(* CoDeSys 2.3.9.41 project: gyps_plant.pro *)
(* Libraries: STANDARD.LIB 4.10.05 13:14:46, IECSFC.LIB 13.4.06 17:51:28, SYSLIBTIME.LIB 20.2.06 15:31:16, SYSTASKINFO.LIB 20.2.06 15:31:38, ANALYZATION.LIB 5.10.99 11:05:06, SYSLIBCALLBACK.LIB 20.2.06 15:31:08, Util.lib 18.5.10 17:14:28 *)

(* PLC configuration (modules and I/O channels)
Fast discrete inputs [I_SIMPLE_INPUT] node 0, in %IB0 out %QB0 {ChannellName = Fast discrete inputs; Filtrationtime = 10000}
  AT %IX0.0 [BitInput] Discrete input 1 {ChannellName = Enter name}
  AT %IX0.1 [BitInput] Discrete input 2 {ChannellName = Enter name}
  AT %IX0.2 [BitInput] Discrete input 3 {ChannellName = Enter name}
  AT %IX0.3 [BitInput] Discrete input 4 {ChannellName = Enter name}
Discrete inputs [ID130] node 1, in %IB1 out %QB1 {ChannellName = Discrete inputs; Filtrationtime_GeneralINP = 0; PinCount = 32}
  AT %IB1.0 [ByteInput] 8 discrete inputs {ChannellName = Enter name}
  AT %IB1.1 [ByteInput] 8 discrete inputs {ChannellName = Enter name}
  AT %IB1.2 [ByteInput] 8 discrete inputs {ChannellName = Enter name}
  AT %IB1.3 [ByteInput] 8 discrete inputs {ChannellName = Enter name}
AT %QX2.0 [BitOutput] Fast discrete output 1 {ChannellName = Enter name}
AT %QX2.1 [BitOutput] Fast discrete output 2 {ChannellName = Enter name}
AT %QX2.2 [BitOutput] Fast discrete output 3 {ChannellName = Enter name}
AT %QX2.3 [BitOutput] Fast discrete output 4 {ChannellName = Enter name}
Discrete outputs [ID131] node 3, in %IB3 out %QB3 {ChannellName = Discrete outputs; SafeValueByte = 0; SafeValueByte = 0; SafeValueByteM = 0; PinCount = 24}
  AT %QB3.0 [ByteOutput] 8 discrete outputs {ChannellName = Enter name}
  AT %QB3.1 [ByteOutput] 8 discrete outputs {ChannellName = Enter name}
  AT %QB3.2 [ByteOutput] 4 discrete outputs {ChannellName = Enter name}
Special input [ID103] node 4, in %IB4 out %QB4 {ChannellName = Special input}
  AT %IX4.0 [BitInput] Special input {ChannellName = Enter name}
Special output [ID104] node 5, in %IB5 out %QB5 {ChannellName = Special output}
  AT %QX5.0 [BitOutput] Special output {ChannellName = Enter name}
ModBus (Master) [MODBUS_MASTER_ID450] node 6, in %IB6 out %QB6 {ChannellName = ModBus (Master); Visibility = No}
  AT %QD6.0 [DWordOutput] Last address {ChannellName = Enter name}
  AT %QW6.1 [WordOutput] Last error {ChannellName = Enter name}
  RS-485-1 [COM1_USART] node 0, in %IB6.0 out %QB6.0 {ChannellName = RS-485-1; CommunicationSpeed = 115200; Parity = NO PARITY CHECK; BitLength = 8 bits; StopLength = One stop bit; InterfaceType = RS485; FrameOriented = RTU; Timeout = 0; Visibility = No}
  Universal Modbus device [ID2000] node 1, in %IB6.1 out %QB6.1 {ChannellName = Universal Modbus device; ModuleIP = 10:0:0:223; ServiceTimeout = 150; TCPport = 502; NetMode = Serial; ModuleSlaveAddress = 8; RequestType = By poll time; PeriodOfService = 10; Visibility = No; RepeatCounter = 0; ByteSequence = Trace_mode}
    AT %QB6.1.0 [ComChannel] Command (0xff - Start) {ChannellName = Enter name}
MV8_0 AT %QW6.1.0.0 [WordOutput] {ChannellName = Enter name}
MV8_1 AT %QW6.1.1.0 [WordOutput] {ChannellName = Enter name}
Universal Modbus device [ID2000] node 2, in %IB6.2 out %QB6.2 {ChannellName = Universal Modbus device; ModuleIP = 10:0:0:223; ServiceTimeout = 150; TCPport = 502; NetMode = Serial; ModuleSlaveAddress = 16; RequestType = By poll time; PeriodOfService = 10; Visibility = No; RepeatCounter = 0; ByteSequence = Trace_mode}
  AT %QB6.2.0 [ComChannel] Command (0xff - Start) {ChannellName = Enter name}
MV16_0 AT %QW6.2.0.0 [WordOutput] {ChannellName = Enter name}
Universal Modbus device [ID2000] node 3, in %IB6.3 out %QB6.3 {ChannellName = Universal Modbus device; ModuleIP = 10:0:0:223; ServiceTimeout = 150; TCPport = 502; NetMode = Serial; ModuleSlaveAddress = 24; RequestType = By poll time; PeriodOfService = 10; Visibility = No; RepeatCounter = 0; ByteSequence = Trace_mode}
  AT %QB6.3.0 [ComChannel] Command (0xff - Start) {ChannellName = Enter name}
MV24_0 AT %QW6.3.0.0 [WordOutput] {ChannellName = Enter name}
MV24_1 AT %QW6.3.1.0 [WordOutput] {ChannellName = Enter name}
Universal Modbus device [ID2000] node 4, in %IB6.4 out %QB6.4 {ChannellName = Universal Modbus device; ModuleIP = 10:0:0:223; ServiceTimeout = 150; TCPport = 502; NetMode = Serial; ModuleSlaveAddress = 32; RequestType = By poll time; PeriodOfService = 10; Visibility = No; RepeatCounter = 0; ByteSequence = Trace_mode}
  AT %QB6.4.0 [ComChannel] Command (0xff - Start) {ChannellName = Enter name}
MU01 AT %QW6.4.0.0 [WordOutput] {ChannellName = Enter name}
MU02 AT %QW6.4.1.0 [WordOutput] {ChannellName = Enter name}
MU03 AT %QW6.4.2.0 [WordOutput] {ChannellName = Enter name}
MU04 AT %QW6.4.3.0 [WordOutput] {ChannellName = Enter name}
MU05 AT %QW6.4.4.0 [WordOutput] {ChannellName = Enter name}
MU06 AT %QW6.4.5.0 [WordOutput] {ChannellName = Enter name}
MU07 AT %QW6.4.6.0 [WordOutput] {ChannellName = Enter name}
MU08 AT %QW6.4.7.0 [WordOutput] {ChannellName = Enter name}
MU09 AT %QW6.4.8.0 [WordOutput] {ChannellName = Enter name}
MU10 AT %QW6.4.9.0 [WordOutput] {ChannellName = Enter name}
MU11 AT %QW6.4.10.0 [WordOutput] {ChannellName = Enter name}
MU12 AT %QW6.4.11.0 [WordOutput] {ChannellName = Enter name}
MU13 AT %QW6.4.12.0 [WordOutput] {ChannellName = Enter name}
MU14 AT %QW6.4.13.0 [WordOutput] {ChannellName = Enter name}
MU15 AT %QW6.4.14.0 [WordOutput] {ChannellName = Enter name}
MU16 AT %QW6.4.15.0 [WordOutput] {ChannellName = Enter name}
MU17 AT %QW6.4.16.0 [WordOutput] {ChannellName = Enter name}
MU18 AT %QW6.4.17.0 [WordOutput] {ChannellName = Enter name}
MU19 AT %QW6.4.18.0 [WordOutput] {ChannellName = Enter name}
MU20 AT %QW6.4.19.0 [WordOutput] {ChannellName = Enter name}
MU21 AT %QW6.4.20.0 [WordOutput] {ChannellName = Enter name}
%MMU22 AT %QW6.4.21.0 [WordOutput] {ChannellName = Enter name}
MU23 AT %QW6.4.22.0 [WordOutput] {ChannellName = Enter name}
MU24 AT %QW6.4.23.0 [WordOutput] {ChannellName = Enter name}
MU25 AT %QW6.4.24.0 [WordOutput] {ChannellName = Enter name}
MU26 AT %QW6.4.25.0 [WordOutput] {ChannellName = Enter name}
MU27 AT %QW6.4.26.0 [WordOutput] {ChannellName = Enter name}
MU28 AT %QW6.4.27.0 [WordOutput] {ChannellName = Enter name}
MU29 AT %QW6.4.28.0 [WordOutput] {ChannellName = Enter name}
MU30 AT %QW6.4.29.0 [WordOutput] {ChannellName = Enter name}
MU31 AT %QW6.4.30.0 [WordOutput] {ChannellName = Enter name}
MU32 AT %QW6.4.31.0 [WordOutput] {ChannellName = Enter name}
AT %QB6.5.0 [ComChannel] Command (0xff - Start) {ChannellName = Enter name}
ELV_CURRENT_4 AT %QD6.5.0.0 [FloatOutput] {ChannellName = Enter name}
SHNK_CURRENT_4 AT %QD6.5.1.0 [FloatOutput] {ChannellName = Enter name}
MILL_SUCTION_4 AT %QD6.5.2.0 [FloatOutput] {ChannellName = Enter name}
SHNK_CURRENT_3 AT %QD6.5.3.0 [FloatOutput] {ChannellName = Enter name}
MILL_SUCTION_3 AT %QD6.5.4.0 [FloatOutput] {ChannellName = Enter name}
Universal Modbus device [ID2000] node 6, in %IB6.6 out %QB6.6 {ChannellName = Universal Modbus device; ModuleIP = 10:0:0:223; ServiceTimeout = 150; TCPport = 502; NetMode = Serial; ModuleSlaveAddress = 48; RequestType = By poll time; PeriodOfService = 10; Visibility = No; RepeatCounter = 0; ByteSequence = Trace_mode}
  AT %QB6.6.0 [ComChannel] Command (0xff - Start) {ChannellName = Enter name}
MV48_0 AT %QW6.6.0.0 [WordOutput] {ChannellName = Enter name}
MV48_1 AT %QW6.6.1.0 [WordOutput] {ChannellName = Enter name}
AT %QB6.7.0 [ComChannel] Command (0xff - Start) {ChannellName = Enter name}
ELV_CUR_0 AT %QD6.7.0.0 [FloatOutput] {ChannellName = Enter name}
SHOK_DROB_1 AT %QD6.7.1.0 [FloatOutput] {ChannellName = Enter name}
SHOK_DROB_2 AT %QD6.7.2.0 [FloatOutput] {ChannellName = Enter name}
ModBus (slave) [MODBUS_ID400] node 7, in %IB7 out %QB7 {ChannellName = ModBus (slave); SlaveIdentificator = 1; Visibility = No}
  Modbus [MODBUS_ID302] node 0, in %IB7.0 out %QB7.0 {ChannellName = Modbus}
    TCP [TCP_ID221] node 0, in %IB7.0.0 out %QB7.0.0 {ChannellName = TCP; RemotePort = 502; Visibility = No}
    TCP [TCP_ID221] node 1, in %IB7.0.1 out %QB7.0.1 {ChannellName = TCP; RemotePort = 503; Visibility = No}
  8 bits [8Bit] node 1, in %IB7.1 out %QB7.1 {ChannellName = 8 bit}
    REG_1_0 AT %QB7.1.0 [ByteOutput] {ChannellName = Enter name}
  8 bits [8Bit] node 2, in %IB7.2 out %QB7.2 {ChannellName = 8 bit}
    REG_1_1 AT %QB7.2.0 [ByteOutput] {ChannellName = Enter name}
  8 bits [8Bit] node 3, in %IB7.3 out %QB7.3 {ChannellName = 8 bit}
    REG_2_0 AT %QB7.3.0 [ByteOutput] {ChannellName = Enter name}
    REG_2_1 AT %QB7.4.0 [ByteOutput] {ChannellName = Enter name}
  8 bits [8Bit] node 5, in %IB7.5 out %QB7.5 {ChannellName = 8 bit}
    REG_3_0 AT %QB7.5.0 [ByteOutput] {ChannellName = Enter name}
  8 bits [8Bit] node 6, in %IB7.6 out %QB7.6 {ChannellName = 8 bit}
    REG_3_1 AT %QB7.6.0 [ByteOutput] {ChannellName = Enter name}
  8 bits [8Bit] node 7, in %IB7.7 out %QB7.7 {ChannellName = 8 bit}
    REG_4_0 AT %QB7.7.0 [ByteOutput] {ChannellName = Enter name}
    REG_4_1 AT %QB7.8.0 [ByteOutput] {ChannellName = Enter name}
    REG_5_0 AT %QB7.9.0 [ByteOutput] {ChannellName = Enter name}
  8 bits [8Bit] node 10, in %IB7.10 out %QB7.10 {ChannellName = 8 bit}
    REG_5_1 AT %QB7.10.0 [ByteOutput] {ChannellName = Enter name}
  8 bits [8Bit] node 11, in %IB7.11 out %QB7.11 {ChannellName = 8 bit}
    REG_6_0 AT %QB7.11.0 [ByteOutput] {ChannellName = Enter name}
    REG_6_1 AT %QB7.12.0 [ByteOutput] {ChannellName = Enter name}
  8 bits [8Bit] node 13, in %IB7.13 out %QB7.13 {ChannellName = 8 bit}
    REG_7_0 AT %QB7.13.0 [ByteOutput] {ChannellName = Enter name}
  8 bits [8Bit] node 14, in %IB7.14 out %QB7.14 {ChannellName = 8 bit}
    REG_7_1 AT %QB7.14.0 [ByteOutput] {ChannellName = Enter name}
  8 bits [8Bit] node 15, in %IB7.15 out %QB7.15 {ChannellName = 8 bit}
    REG_8_0 AT %QB7.15.0 [ByteOutput] {ChannellName = Enter name}
    REG_8_1 AT %QB7.16.0 [ByteOutput] {ChannellName = Enter name}
  8 bits [8Bit] node 17, in %IB7.17 out %QB7.17 {ChannellName = 8 bit}
    REG_9_0 AT %QB7.17.0 [ByteOutput] {ChannellName = Enter name}
  8 bits [8Bit] node 18, in %IB7.18 out %QB7.18 {ChannellName = 8 bit}
    REG_9_1 AT %QB7.18.0 [ByteOutput] {ChannellName = Enter name}
  8 bits [8Bit] node 19, in %IB7.19 out %QB7.19 {ChannellName = 8 bit}
    REG_10_0 AT %QB7.19.0 [ByteOutput] {ChannellName = Enter name}
    REG_10_1 AT %QB7.20.0 [ByteOutput] {ChannellName = Enter name}
  8 bits [8Bit] node 21, in %IB7.21 out %QB7.21 {ChannellName = 8 bit}
    REG_11_0 AT %QB7.21.0 [ByteOutput] {ChannellName = Enter name}
  8 bits [8Bit] node 22, in %IB7.22 out %QB7.22 {ChannellName = 8 bit}
    REG_11_1 AT %QB7.22.0 [ByteOutput] {ChannellName = Enter name}
  8 bits [8Bit] node 23, in %IB7.23 out %QB7.23 {ChannellName = 8 bit}
    REG_12_0 AT %QB7.23.0 [ByteOutput] {ChannellName = Enter name}
    REG_12_1 AT %QB7.24.0 [ByteOutput] {ChannellName = Enter name}
REG_13_ELV_CURRENT_4 AT %QD7.25.0 [FloatOutput] {ChannellName = Enter name}
REG_15_SHNK_CURRENT_4 AT %QD7.26.0 [FloatOutput] {ChannellName = Enter name}
REG_17_MILL_SUCTION_4 AT %QD7.27.0 [FloatOutput] {ChannellName = Enter name}
REG_19_SHNK_CURRENT_3 AT %QD7.28.0 [FloatOutput] {ChannellName = Enter name}
REG_21_MILL_SUCTION_3 AT %QD7.29.0 [FloatOutput] {ChannellName = Enter name}
REG_23_ELV_CUR_0 AT %QD7.30.0 [FloatOutput] {ChannellName = Enter name}
REG_25_SHOK_DROB_1 AT %QD7.31.0 [FloatOutput] {ChannellName = Enter name}
REG_27_SHOK_DROB_2 AT %QD7.32.0 [FloatOutput] {ChannellName = Enter name}
REG_29 AT %QD7.33.0 [FloatOutput] {ChannellName = Enter name}
REG_31 AT %QD7.34.0 [FloatOutput] {ChannellName = Enter name}
REG_33 AT %QD7.35.0 [FloatOutput] {ChannellName = Enter name}
REG_35 AT %QD7.36.0 [FloatOutput] {ChannellName = Enter name}
AT %QD8.0 [DWordOutput] Last address {ChannellName = Enter name}
AT %QW8.1 [WordOutput] Last error {ChannellName = Enter name}
RS-485-2 [COM3_USART] node 0, in %IB8.0 out %QB8.0 {ChannellName = RS-485-2; CommunicationSpeed = 115200; Parity = NO PARITY CHECK; BitLength = 8 bits; StopLength = One stop bit; InterfaceType = RS485; FrameOriented = RTU; Timeout = 0; Visibility = No}
Universal Modbus device [ID2000] node 1, in %IB8.1 out %QB8.1 {ChannellName = Universal Modbus device; ModuleIP = 10:0:0:223; ServiceTimeout = 150; TCPport = 502; NetMode = Serial; ModuleSlaveAddress = 1; RequestType = By poll time; PeriodOfService = 100; Visibility = No; RepeatCounter = 0; ByteSequence = Trace_mode}
  AT %QB8.1.0 [ComChannel] Command (0xff - Start) {ChannellName = Enter name}
CONV_PANEL_3 AT %QW8.1.0.0 [WordOutput] {ChannellName = Enter name}
CONV_FREQ_3 AT %QW8.1.1.0 [WordOutput] {ChannellName = Enter name}
CONV_CURRENT_3 AT %QW8.1.2.0 [WordOutput] {ChannellName = Enter name}
CONV_SET_FREQ_3 AT %QW8.1.3.0 [WordOutput] {ChannellName = Enter name}
AT %QB8.2.0 [ComChannel] Command (0xff - Start)
FAN_PANEL_3 AT %QW8.2.0.0 [WordOutput] {ChannellName = Enter name}
FAN_FREQ_3 AT %QW8.2.1.0 [WordOutput] {ChannellName = Enter name}
FAN_CURRENT_3 AT %QW8.2.2.0 [WordOutput] {ChannellName = Enter name}
FAN_SET_FREQ_3 AT %QW8.2.3.0 [WordOutput] {ChannellName = Enter name}
AT %QB8.3.0 [ComChannel] Command (0xff - Start) {ChannellName = Enter name}
MILL_PANEL_3 AT %QW8.3.0.0 [WordOutput] {ChannellName = Enter name}
MILL_FREQ_3 AT %QW8.3.1.0 [WordOutput] {ChannellName = Enter name}
MILL_CURRENT_3 AT %QW8.3.2.0 [WordOutput] {ChannellName = Enter name}
MILL_SET_FREQ_3 AT %QW8.3.3.0 [WordOutput] {ChannellName = Enter name}
AT %QB8.4.0 [ComChannel] Command (0xff - Start) {ChannellName = Enter name}
SEP_PANEL_3 AT %QW8.4.0.0 [WordOutput] {ChannellName = Enter name}
SEP_FREQ_3 AT %QW8.4.1.0 [WordOutput] {ChannellName = Enter name}
SEP_CURRENT_3 AT %QW8.4.2.0 [WordOutput] {ChannellName = Enter name}
SEP_SET_FREQ_3 AT %QW8.4.3.0 [WordOutput] {ChannellName = Enter name}
AT %QB8.5.0 [ComChannel] Command (0xff - Start) {ChannellName = Enter name}
CONV_PANEL_4 AT %QW8.5.0.0 [WordOutput] {ChannellName = Enter name}
CONV_FREQ_4 AT %QW8.5.1.0 [WordOutput] {ChannellName = Enter name}
CONV_CURRENT_4 AT %QW8.5.2.0 [WordOutput] {ChannellName = Enter name}
CONV_SET_FREQ_4 AT %QW8.5.3.0 [WordOutput] {ChannellName = Enter name}
AT %QB8.6.0 [ComChannel] Command (0xff - Start)
FAN_PANEL_4 AT %QW8.6.0.0 [WordOutput] {ChannellName = Enter name}
FAN_FREQ_4 AT %QW8.6.1.0 [WordOutput] {ChannellName = Enter name}
FAN_CURRENT_4 AT %QW8.6.2.0 [WordOutput] {ChannellName = Enter name}
FAN_SET_FREQ_4 AT %QW8.6.3.0 [WordOutput] {ChannellName = Enter name}
AT %QB8.7.0 [ComChannel] Command (0xff - Start) {ChannellName = Enter name}
MILL_PANEL_4 AT %QW8.7.0.0 [WordOutput] {ChannellName = Enter name}
MILL_FREQ_4 AT %QW8.7.1.0 [WordOutput] {ChannellName = Enter name}
MILL_CURRENT_4 AT %QW8.7.2.0 [WordOutput] {ChannellName = Enter name}
MILL_SET_FREQ_4 AT %QW8.7.3.0 [WordOutput] {ChannellName = Enter name}
AT %QB8.8.0 [ComChannel] Command (0xff - Start) {ChannellName = Enter name}
SEP_PANEL_4 AT %QW8.8.0.0 [WordOutput] {ChannellName = Enter name}
SEP_FREQ_4 AT %QW8.8.1.0 [WordOutput] {ChannellName = Enter name}
SEP_CURRENT_4 AT %QW8.8.2.0 [WordOutput] {ChannellName = Enter name}
SEP_SET_FREQ_4 AT %QW8.8.3.0 [WordOutput] {ChannellName = Enter name}
*)

(* Global variable list: Global_Variables *)
VAR_GLOBAL
	kvitVaqt : TIME := T#60s;
	tpKVIT : TP;
	HORN_RESET_0 : BOOL;
	(*MU 32 DISCRET OUTPUT*)
	ELV_RUN : BOOL;			(*DO01*)
	SHNK_RUN_4  : BOOL;		(*DO02*)
	SHNK_SKL_RUN_4  : BOOL;	(*DO03*)
	STAR_RUN_41  : BOOL;		(*DO04*)
	STAR_RUN_42  : BOOL;		(*DO05*)
	SEPR_RUN_4  : BOOL;		(*DO06*)
	OIL_ST_RUN_4  : BOOL;		(*DO07*)
	MILL_RUN_4  : BOOL;		(*DO08*)
	FAN_RUN_4  : BOOL;		(*DO09*)
	CONV_RUN_4  : BOOL;		(*DO10*)
	VIBR_RUN_4  : BOOL;		(*DO11*)
	VALV_RUN_4 : BOOL;		(*DO12*)
	HORN_RUN_4 : BOOL; 		(*DO13*)

	(*ELV_RUN_3 :  BOOL ; 		DO17*)
	SHNK_RUN_3 :  BOOL ; 		(*DO18*)
	SHNK_SKL_RUN_3 :  BOOL ; (*DO19*)
	STAR_RUN_31 :  BOOL ;  	(*DO20*)
	STAR_RUN_32 :  BOOL ;  	(*DO21*)
	SEPR_RUN_3 :  BOOL ;  		(*DO22*)
	OIL_ST_RUN_3 :  BOOL ;  	(*DO23*)
	MILL_RUN_3 :  BOOL ;  		(*DO24*)
	FAN_RUN_3 :  BOOL ;  		(*DO25*)
	CONV_RUN_3 :  BOOL ; 		(*DO26*)
	VIBR_RUN_3 :  BOOL ;  		(*DO27*)
	VALV_RUN_3 :  BOOL ;  		(*DO28*)
	HORN_RUN_3 :  BOOL ; 		(*DO29*)
	(*MU 32 DISCRET OUTPUT*)
	(*MV 24 DISCRET INPUT*)
	ELV_KM  : BOOL;				(*DI01*)
	SHNK_KM_4  : BOOL;			(*DI02*)
	SHNK_SKL_KM_4  : BOOL;		(*DI03*)
	STAR_KM_41  : BOOL;			(*DI04*)
	STAR_KM_42  : BOOL;			(*DI05*)
	SEPR_KM_4  : BOOL;			(*DI06*)
	OIL_ST_KM_4  : BOOL;			(*DI07*)
	MILL_KM_4  : BOOL;			(*DI08*)
	MATER_FULL_4  : BOOL;		(*DI09*)
	FAN_KM_4  : BOOL;				(*DI10*)
	CONV_KM_4  : BOOL;			(*DI11*)
	VIBR_KM_4  : BOOL;			(*DI12*)

				(*DI17*)
	SHNK_KM_3  : BOOL;			(*DI18*)
	SHNK_SKL_KM_3  : BOOL;		(*DI19*)
	STAR_KM_31  : BOOL;			(*DI20*)
	STAR_KM_32  : BOOL;			(*DI21*)
	SEPR_KM_3  : BOOL;			(*DI22*)
	OIL_ST_KM_3  : BOOL;			(*DI23*)
	MILL_KM_3  : BOOL;			(*DI24*)
	MATER_FULL_3  : BOOL;		(*DI25*)
	FAN_KM_3  : BOOL;				(*DI26*)
	CONV_KM_3  : BOOL;			(*DI27*)
	VIBR_KM_3  : BOOL;			(*DI28*)
	CONTR_PHASE_1_2 : BOOL;
	(*MV 24 DISCRET INPUT*)
	(*MV 16 DISCRET INPUT*)
	ELV_STOP_3  : BOOL;			(*DI01*)
	SHNK_STOP_3  : BOOL;			(*DI02*)
	SHNK_SKL_STOP_3  : BOOL;	(*DI03*)
	STAR_STOP_31  : BOOL;		(*DI04*)
	STAR_STOP_32  : BOOL;		(*DI05*)
	SEPR_STOP_3  : BOOL;			(*DI06*)
	OIL_ST_STOP_3  : BOOL;		(*DI07*)
	MILL_STOP_3  : BOOL;			(*DI08*)
	FAN_STOP_3  : BOOL;			(*DI09*)
	CONV_STOP_3  : BOOL;			(*DI10*)
	VIBR_STOP_3  : BOOL;			(*DI11*)

	ELV_START_3 : BOOL;			(*DI17*)
	SHNK_START_3 : BOOL;			(*DI18*)
	SHNK_SKL_START_3 : BOOL;	(*DI19*)
	STAR_START_31 : BOOL;		(*DI20*)
	STAR_START_32 : BOOL;		(*DI21*)
	SEPR_START_3 : BOOL;			(*DI22*)
	OIL_ST_START_3 : BOOL;		(*DI23*)
	MILL_START_3 : BOOL;			(*DI24*)
	FAN_START_3 : BOOL;			(*DI25*)
	CONV_START_3 : BOOL;		(*DI26*)
	VIBR_START_3 : BOOL;			(*DI27*)
	(*MV 16 DISCRET INPUT*)
	(*MV 08 DISCRET INPUT*)
	ELV_STOP_4  : BOOL;			(*DI01*)
	SHNK_STOP_4  : BOOL;			(*DI02*)
	SHNK_SKL_STOP_4  : BOOL;	(*DI03*)
	STAR_STOP_41  : BOOL;		(*DI04*)
	STAR_STOP_42  : BOOL;		(*DI05*)
	SEPR_STOP_4  : BOOL;			(*DI06*)
	OIL_ST_STOP_4  : BOOL;		(*DI07*)
	MILL_STOP_4  : BOOL;			(*DI08*)
	FAN_STOP_4  : BOOL;			(*DI09*)
	CONV_STOP_4  : BOOL;			(*DI10*)
	VIBR_STOP_4  : BOOL;			(*DI11*)

	ELV_START_4  : BOOL;			(*DI17*)
	SHNK_START_4  : BOOL;		(*DI18*)
	SHNK_SKL_START_4  : BOOL;	(*DI19*)
	STAR_START_41  : BOOL;		(*DI20*)
	STAR_START_42  : BOOL;		(*DI21*)
	SEPR_START_4  : BOOL;		(*DI22*)
	OIL_ST_START_4  : BOOL;		(*DI23*)
	MILL_START_4  : BOOL;			(*DI24*)
	FAN_START_4  : BOOL;			(*DI25*)
	CONV_START_4  : BOOL;			(*DI26*)
	VIBR_START_4  : BOOL;			(*DI27*)
	(*MV 08 DISCRET INPUT*)
END_VAR

(* Global variable list: mb_drob_in *)
VAR_GLOBAL
	MB_EMER_STOP_0 : BOOL;
	MB_MANUAL_ELV_0 : BOOL;
	MB_AUTO_ELV_0 : BOOL;
	MB_RESET_0 : BOOL;
	MB_ELV_STOP_0 : BOOL;
	MB_ELV_START_0 : BOOL;
	MB_SHOK_DROB_STOP_1 : BOOL;
	MB_SHOK_DROB_START_1 : BOOL;
	MB_SHOK_DROB_STOP_2 : BOOL;
	MB_SHOK_DROB_START_2 : BOOL;
	MB_CONV_STOP_0 : BOOL;
	MB_CONV_START_0 : BOOL;
	(****RESERV CONV ***)
	(***RESERV CONV****)
	MB_ELV_KM_0 : BOOL;
	MB_SHOK_DROB_KM_1 : BOOL;
	MB_SHOK_DROB_KM_2 : BOOL;
	MB_CONV_KM_0 : BOOL;
	(** RESERV KM CONV **)
	MB_TANK_MAX_0 : BOOL;
	MB_TANK_MIDLE_0 : BOOL;
	MB_TANK_MIN_0 : BOOL;


END_VAR

(* POU PLC_PRG, ST *)
PROGRAM PLC_PRG
VAR
END_VAR
main();
ALARMS();
RESET_ALRM();
TRANSLATE();
DROBILKA();
END_PROGRAM

(* POU main, LD *)
PROGRAM main
VAR
	MAH_YET3 : BOOL;
	VAQT : TIME := T#10s;
       VAQT1: TIME := T#4s;
       VAQT2 : TIME := T#6s;
      VAQT3 : TIME := T#6s;
	vaqtInduc : WORD := 15;
	VIBRATOR3_T: BOOL;
	TON1: TON;
	TON2: TON;
	OUT: BOOL;
	IND1: INDUKTIV;
	IND2: INDUKTIV;


	STOP: BOOL;
	CHIQSH: BOOL;
	PUSK: BOOL;
	MAH_YET4: BOOL;
	VIBRATOR4_T: BOOL;
	induk: BOOL;

	ALR_ELEV1: BOOL;
	ALR_ELEV2: BOOL;
	ALR_ELEV3: BOOL;
	ALR_ELEV4: BOOL;
	IND_ELV_1: INDUKTIV;
	IND_SHNK_3: INDUKTIV;
	IND_SHNK_4: INDUKTIV;
	IND_SHNK_SKL_4: INDUKTIV;
	IND_SEPR_4: INDUKTIV;
	IND_MILL_3: INDUKTIV;
	IND_MILL_4: INDUKTIV;

END_VAR
VAR (* helpers for the ST form of the networks *)
	_p1 : BOOL;
	_p2 : BOOL;
	_p3 : BOOL;
	_p4 : BOOL;
	_p5 : BOOL;
	_p6 : BOOL;
	_p7 : BOOL;
END_VAR
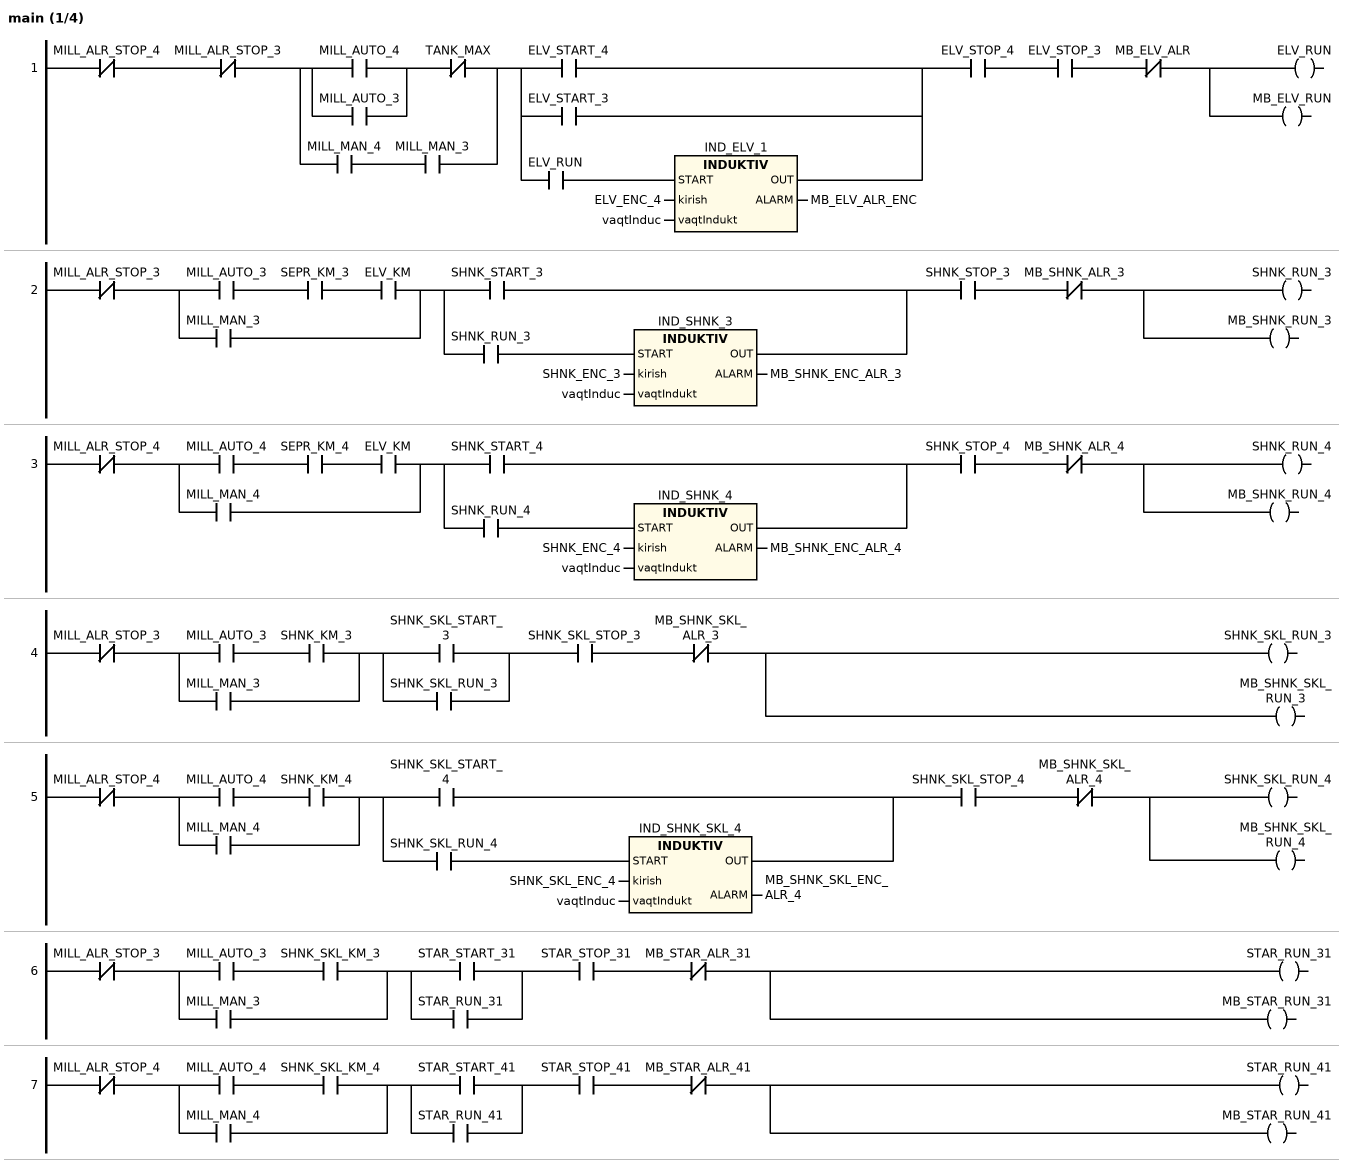
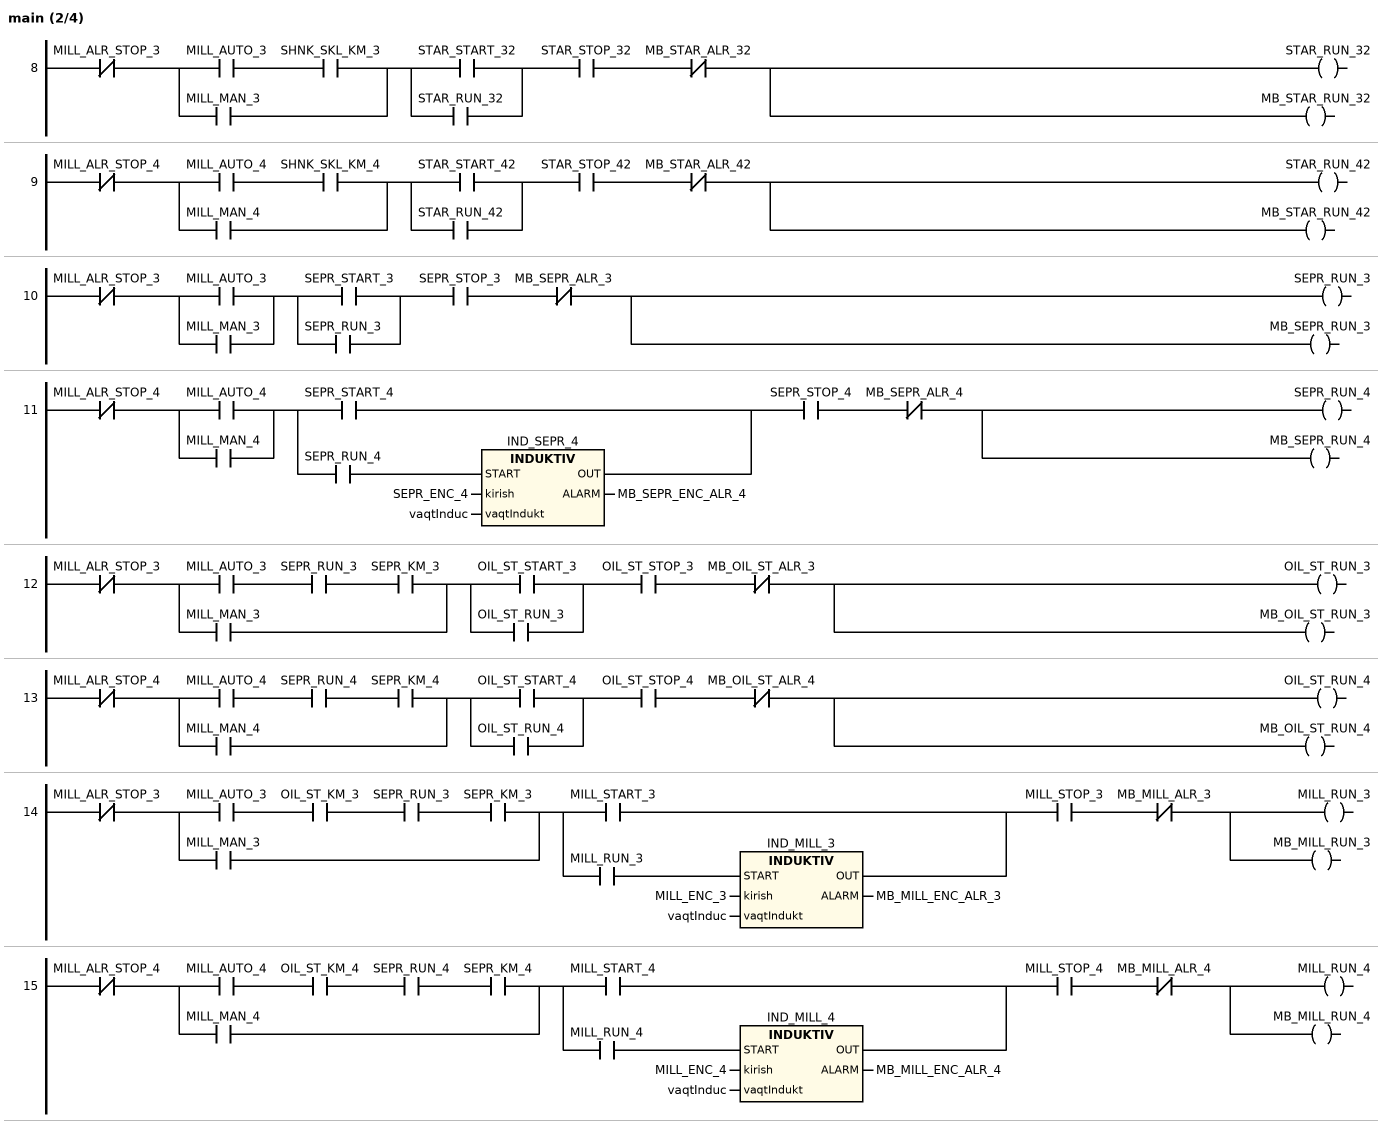
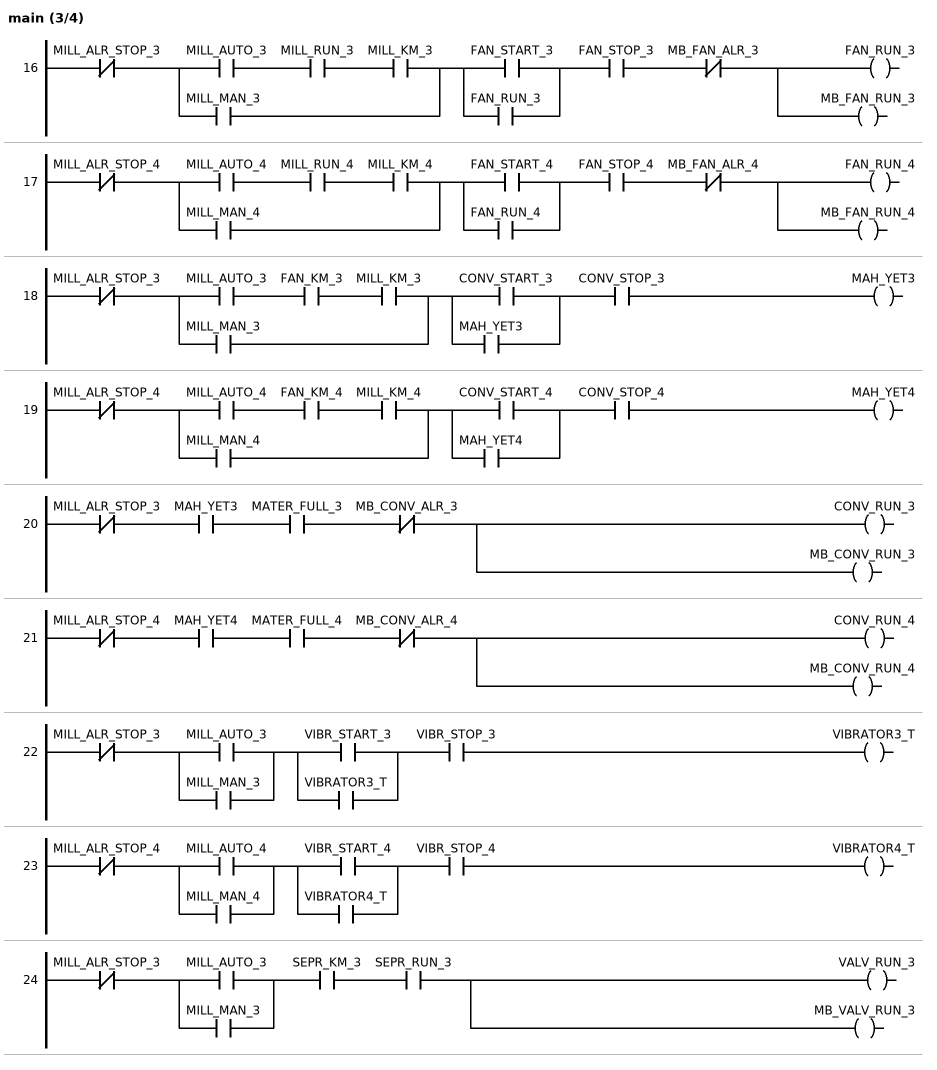
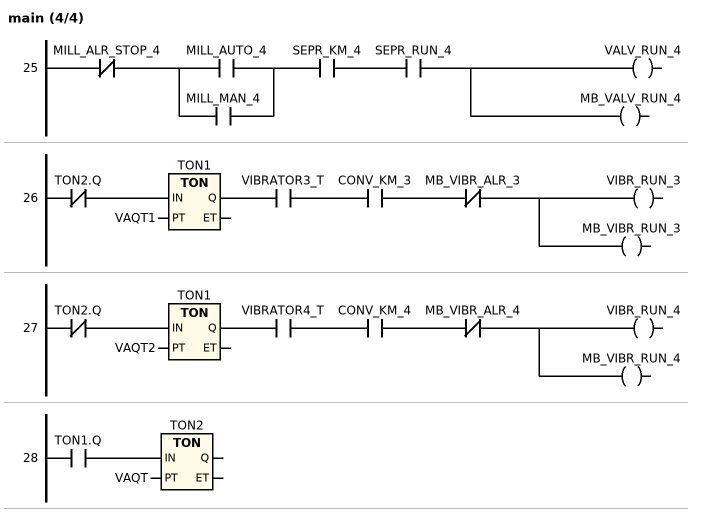
_LD_ (* Ladder Diagram *)
NETWORK 1
	[/MILL_ALR_STOP_4] - [/MILL_ALR_STOP_3] - { { [MILL_AUTO_4] | [MILL_AUTO_3] } - [/TANK_MAX] | [MILL_MAN_4] - [MILL_MAN_3] } - { [ELV_START_4] | [ELV_START_3] | [ELV_RUN] - IND_ELV_1:INDUKTIV(START: *, kirish: ELV_ENC_4, vaqtIndukt: vaqtInduc, ALARM => MB_ELV_ALR_ENC) } - [ELV_STOP_4] - [ELV_STOP_3] - [/MB_ELV_ALR] --- (ELV_RUN) (MB_ELV_RUN)
NETWORK 2
	[/MILL_ALR_STOP_3] - { [MILL_AUTO_3] - [SEPR_KM_3] - [ELV_KM] | [MILL_MAN_3] } - { [SHNK_START_3] | [SHNK_RUN_3] - IND_SHNK_3:INDUKTIV(START: *, kirish: SHNK_ENC_3, vaqtIndukt: vaqtInduc, ALARM => MB_SHNK_ENC_ALR_3) } - [SHNK_STOP_3] - [/MB_SHNK_ALR_3] --- (SHNK_RUN_3) (MB_SHNK_RUN_3)
NETWORK 3
	[/MILL_ALR_STOP_4] - { [MILL_AUTO_4] - [SEPR_KM_4] - [ELV_KM] | [MILL_MAN_4] } - { [SHNK_START_4] | [SHNK_RUN_4] - IND_SHNK_4:INDUKTIV(START: *, kirish: SHNK_ENC_4, vaqtIndukt: vaqtInduc, ALARM => MB_SHNK_ENC_ALR_4) } - [SHNK_STOP_4] - [/MB_SHNK_ALR_4] --- (SHNK_RUN_4) (MB_SHNK_RUN_4)
NETWORK 4
	[/MILL_ALR_STOP_3] - { [MILL_AUTO_3] - [SHNK_KM_3] | [MILL_MAN_3] } - { [SHNK_SKL_START_3] | [SHNK_SKL_RUN_3] } - [SHNK_SKL_STOP_3] - [/MB_SHNK_SKL_ALR_3] --- (SHNK_SKL_RUN_3) (MB_SHNK_SKL_RUN_3)
NETWORK 5
	[/MILL_ALR_STOP_4] - { [MILL_AUTO_4] - [SHNK_KM_4] | [MILL_MAN_4] } - { [SHNK_SKL_START_4] | [SHNK_SKL_RUN_4] - IND_SHNK_SKL_4:INDUKTIV(START: *, kirish: SHNK_SKL_ENC_4, vaqtIndukt: vaqtInduc, ALARM => MB_SHNK_SKL_ENC_ALR_4) } - [SHNK_SKL_STOP_4] - [/MB_SHNK_SKL_ALR_4] --- (SHNK_SKL_RUN_4) (MB_SHNK_SKL_RUN_4)
NETWORK 6
	[/MILL_ALR_STOP_3] - { [MILL_AUTO_3] - [SHNK_SKL_KM_3] | [MILL_MAN_3] } - { [STAR_START_31] | [STAR_RUN_31] } - [STAR_STOP_31] - [/MB_STAR_ALR_31] --- (STAR_RUN_31) (MB_STAR_RUN_31)
NETWORK 7
	[/MILL_ALR_STOP_4] - { [MILL_AUTO_4] - [SHNK_SKL_KM_4] | [MILL_MAN_4] } - { [STAR_START_41] | [STAR_RUN_41] } - [STAR_STOP_41] - [/MB_STAR_ALR_41] --- (STAR_RUN_41) (MB_STAR_RUN_41)
NETWORK 8
	[/MILL_ALR_STOP_3] - { [MILL_AUTO_3] - [SHNK_SKL_KM_3] | [MILL_MAN_3] } - { [STAR_START_32] | [STAR_RUN_32] } - [STAR_STOP_32] - [/MB_STAR_ALR_32] --- (STAR_RUN_32) (MB_STAR_RUN_32)
NETWORK 9
	[/MILL_ALR_STOP_4] - { [MILL_AUTO_4] - [SHNK_SKL_KM_4] | [MILL_MAN_4] } - { [STAR_START_42] | [STAR_RUN_42] } - [STAR_STOP_42] - [/MB_STAR_ALR_42] --- (STAR_RUN_42) (MB_STAR_RUN_42)
NETWORK 10
	[/MILL_ALR_STOP_3] - { [MILL_AUTO_3] | [MILL_MAN_3] } - { [SEPR_START_3] | [SEPR_RUN_3] } - [SEPR_STOP_3] - [/MB_SEPR_ALR_3] --- (SEPR_RUN_3) (MB_SEPR_RUN_3)
NETWORK 11
	[/MILL_ALR_STOP_4] - { [MILL_AUTO_4] | [MILL_MAN_4] } - { [SEPR_START_4] | [SEPR_RUN_4] - IND_SEPR_4:INDUKTIV(START: *, kirish: SEPR_ENC_4, vaqtIndukt: vaqtInduc, ALARM => MB_SEPR_ENC_ALR_4) } - [SEPR_STOP_4] - [/MB_SEPR_ALR_4] --- (SEPR_RUN_4) (MB_SEPR_RUN_4)
NETWORK 12
	[/MILL_ALR_STOP_3] - { [MILL_AUTO_3] - [SEPR_RUN_3] - [SEPR_KM_3] | [MILL_MAN_3] } - { [OIL_ST_START_3] | [OIL_ST_RUN_3] } - [OIL_ST_STOP_3] - [/MB_OIL_ST_ALR_3] --- (OIL_ST_RUN_3) (MB_OIL_ST_RUN_3)
NETWORK 13
	[/MILL_ALR_STOP_4] - { [MILL_AUTO_4] - [SEPR_RUN_4] - [SEPR_KM_4] | [MILL_MAN_4] } - { [OIL_ST_START_4] | [OIL_ST_RUN_4] } - [OIL_ST_STOP_4] - [/MB_OIL_ST_ALR_4] --- (OIL_ST_RUN_4) (MB_OIL_ST_RUN_4)
NETWORK 14
	[/MILL_ALR_STOP_3] - { [MILL_AUTO_3] - [OIL_ST_KM_3] - [SEPR_RUN_3] - [SEPR_KM_3] | [MILL_MAN_3] } - { [MILL_START_3] | [MILL_RUN_3] - IND_MILL_3:INDUKTIV(START: *, kirish: MILL_ENC_3, vaqtIndukt: vaqtInduc, ALARM => MB_MILL_ENC_ALR_3) } - [MILL_STOP_3] - [/MB_MILL_ALR_3] --- (MILL_RUN_3) (MB_MILL_RUN_3)
NETWORK 15
	[/MILL_ALR_STOP_4] - { [MILL_AUTO_4] - [OIL_ST_KM_4] - [SEPR_RUN_4] - [SEPR_KM_4] | [MILL_MAN_4] } - { [MILL_START_4] | [MILL_RUN_4] - IND_MILL_4:INDUKTIV(START: *, kirish: MILL_ENC_4, vaqtIndukt: vaqtInduc, ALARM => MB_MILL_ENC_ALR_4) } - [MILL_STOP_4] - [/MB_MILL_ALR_4] --- (MILL_RUN_4) (MB_MILL_RUN_4)
NETWORK 16
	[/MILL_ALR_STOP_3] - { [MILL_AUTO_3] - [MILL_RUN_3] - [MILL_KM_3] | [MILL_MAN_3] } - { [FAN_START_3] | [FAN_RUN_3] } - [FAN_STOP_3] - [/MB_FAN_ALR_3] --- (FAN_RUN_3) (MB_FAN_RUN_3)
NETWORK 17
	[/MILL_ALR_STOP_4] - { [MILL_AUTO_4] - [MILL_RUN_4] - [MILL_KM_4] | [MILL_MAN_4] } - { [FAN_START_4] | [FAN_RUN_4] } - [FAN_STOP_4] - [/MB_FAN_ALR_4] --- (FAN_RUN_4) (MB_FAN_RUN_4)
NETWORK 18
	[/MILL_ALR_STOP_3] - { [MILL_AUTO_3] - [FAN_KM_3] - [MILL_KM_3] | [MILL_MAN_3] } - { [CONV_START_3] | [MAH_YET3] } - [CONV_STOP_3] --- (MAH_YET3)
NETWORK 19
	[/MILL_ALR_STOP_4] - { [MILL_AUTO_4] - [FAN_KM_4] - [MILL_KM_4] | [MILL_MAN_4] } - { [CONV_START_4] | [MAH_YET4] } - [CONV_STOP_4] --- (MAH_YET4)
NETWORK 20
	[/MILL_ALR_STOP_3] - [MAH_YET3] - [MATER_FULL_3] - [/MB_CONV_ALR_3] --- (CONV_RUN_3) (MB_CONV_RUN_3)
NETWORK 21
	[/MILL_ALR_STOP_4] - [MAH_YET4] - [MATER_FULL_4] - [/MB_CONV_ALR_4] --- (CONV_RUN_4) (MB_CONV_RUN_4)
NETWORK 22
	[/MILL_ALR_STOP_3] - { [MILL_AUTO_3] | [MILL_MAN_3] } - { [VIBR_START_3] | [VIBRATOR3_T] } - [VIBR_STOP_3] --- (VIBRATOR3_T)
NETWORK 23
	[/MILL_ALR_STOP_4] - { [MILL_AUTO_4] | [MILL_MAN_4] } - { [VIBR_START_4] | [VIBRATOR4_T] } - [VIBR_STOP_4] --- (VIBRATOR4_T)
NETWORK 24
	[/MILL_ALR_STOP_3] - { [MILL_AUTO_3] | [MILL_MAN_3] } - [SEPR_KM_3] - [SEPR_RUN_3] --- (VALV_RUN_3) (MB_VALV_RUN_3)
NETWORK 25
	[/MILL_ALR_STOP_4] - { [MILL_AUTO_4] | [MILL_MAN_4] } - [SEPR_KM_4] - [SEPR_RUN_4] --- (VALV_RUN_4) (MB_VALV_RUN_4)
NETWORK 26
	[/TON2.Q] - TON1:TON(IN: *, PT: VAQT1) - [VIBRATOR3_T] - [CONV_KM_3] - [/MB_VIBR_ALR_3] --- (VIBR_RUN_3) (MB_VIBR_RUN_3)
NETWORK 27
	[/TON2.Q] - TON1:TON(IN: *, PT: VAQT2) - [VIBRATOR4_T] - [CONV_KM_4] - [/MB_VIBR_ALR_4] --- (VIBR_RUN_4) (MB_VIBR_RUN_4)
NETWORK 28
	[TON1.Q] - TON2:TON(IN: *, PT: VAQT)
_END_LD_
(* the same logic as Structured Text *)
(* Network 1 *)
_p1 := NOT MILL_ALR_STOP_4 AND NOT MILL_ALR_STOP_3 AND ((MILL_AUTO_4 OR MILL_AUTO_3) AND NOT TANK_MAX OR MILL_MAN_4 AND MILL_MAN_3);
IND_ELV_1(START := _p1 AND ELV_RUN, kirish := ELV_ENC_4, vaqtIndukt := vaqtInduc);
MB_ELV_ALR_ENC := IND_ELV_1.ALARM;
ELV_RUN := (_p1 AND ELV_START_4 OR _p1 AND ELV_START_3 OR IND_ELV_1.OUT) AND ELV_STOP_4 AND ELV_STOP_3 AND NOT MB_ELV_ALR;
MB_ELV_RUN := ELV_RUN;
(* Network 2 *)
_p2 := NOT MILL_ALR_STOP_3 AND (MILL_AUTO_3 AND SEPR_KM_3 AND ELV_KM OR MILL_MAN_3);
IND_SHNK_3(START := _p2 AND SHNK_RUN_3, kirish := SHNK_ENC_3, vaqtIndukt := vaqtInduc);
MB_SHNK_ENC_ALR_3 := IND_SHNK_3.ALARM;
SHNK_RUN_3 := (_p2 AND SHNK_START_3 OR IND_SHNK_3.OUT) AND SHNK_STOP_3 AND NOT MB_SHNK_ALR_3;
MB_SHNK_RUN_3 := SHNK_RUN_3;
(* Network 3 *)
_p3 := NOT MILL_ALR_STOP_4 AND (MILL_AUTO_4 AND SEPR_KM_4 AND ELV_KM OR MILL_MAN_4);
IND_SHNK_4(START := _p3 AND SHNK_RUN_4, kirish := SHNK_ENC_4, vaqtIndukt := vaqtInduc);
MB_SHNK_ENC_ALR_4 := IND_SHNK_4.ALARM;
SHNK_RUN_4 := (_p3 AND SHNK_START_4 OR IND_SHNK_4.OUT) AND SHNK_STOP_4 AND NOT MB_SHNK_ALR_4;
MB_SHNK_RUN_4 := SHNK_RUN_4;
(* Network 4 *)
SHNK_SKL_RUN_3 := NOT MILL_ALR_STOP_3 AND (MILL_AUTO_3 AND SHNK_KM_3 OR MILL_MAN_3) AND (SHNK_SKL_START_3 OR SHNK_SKL_RUN_3) AND SHNK_SKL_STOP_3 AND NOT MB_SHNK_SKL_ALR_3;
MB_SHNK_SKL_RUN_3 := SHNK_SKL_RUN_3;
(* Network 5 *)
_p4 := NOT MILL_ALR_STOP_4 AND (MILL_AUTO_4 AND SHNK_KM_4 OR MILL_MAN_4);
IND_SHNK_SKL_4(START := _p4 AND SHNK_SKL_RUN_4, kirish := SHNK_SKL_ENC_4, vaqtIndukt := vaqtInduc);
MB_SHNK_SKL_ENC_ALR_4 := IND_SHNK_SKL_4.ALARM;
SHNK_SKL_RUN_4 := (_p4 AND SHNK_SKL_START_4 OR IND_SHNK_SKL_4.OUT) AND SHNK_SKL_STOP_4 AND NOT MB_SHNK_SKL_ALR_4;
MB_SHNK_SKL_RUN_4 := SHNK_SKL_RUN_4;
(* Network 6 *)
STAR_RUN_31 := NOT MILL_ALR_STOP_3 AND (MILL_AUTO_3 AND SHNK_SKL_KM_3 OR MILL_MAN_3) AND (STAR_START_31 OR STAR_RUN_31) AND STAR_STOP_31 AND NOT MB_STAR_ALR_31;
MB_STAR_RUN_31 := STAR_RUN_31;
(* Network 7 *)
STAR_RUN_41 := NOT MILL_ALR_STOP_4 AND (MILL_AUTO_4 AND SHNK_SKL_KM_4 OR MILL_MAN_4) AND (STAR_START_41 OR STAR_RUN_41) AND STAR_STOP_41 AND NOT MB_STAR_ALR_41;
MB_STAR_RUN_41 := STAR_RUN_41;
(* Network 8 *)
STAR_RUN_32 := NOT MILL_ALR_STOP_3 AND (MILL_AUTO_3 AND SHNK_SKL_KM_3 OR MILL_MAN_3) AND (STAR_START_32 OR STAR_RUN_32) AND STAR_STOP_32 AND NOT MB_STAR_ALR_32;
MB_STAR_RUN_32 := STAR_RUN_32;
(* Network 9 *)
STAR_RUN_42 := NOT MILL_ALR_STOP_4 AND (MILL_AUTO_4 AND SHNK_SKL_KM_4 OR MILL_MAN_4) AND (STAR_START_42 OR STAR_RUN_42) AND STAR_STOP_42 AND NOT MB_STAR_ALR_42;
MB_STAR_RUN_42 := STAR_RUN_42;
(* Network 10 *)
SEPR_RUN_3 := NOT MILL_ALR_STOP_3 AND (MILL_AUTO_3 OR MILL_MAN_3) AND (SEPR_START_3 OR SEPR_RUN_3) AND SEPR_STOP_3 AND NOT MB_SEPR_ALR_3;
MB_SEPR_RUN_3 := SEPR_RUN_3;
(* Network 11 *)
_p5 := NOT MILL_ALR_STOP_4 AND (MILL_AUTO_4 OR MILL_MAN_4);
IND_SEPR_4(START := _p5 AND SEPR_RUN_4, kirish := SEPR_ENC_4, vaqtIndukt := vaqtInduc);
MB_SEPR_ENC_ALR_4 := IND_SEPR_4.ALARM;
SEPR_RUN_4 := (_p5 AND SEPR_START_4 OR IND_SEPR_4.OUT) AND SEPR_STOP_4 AND NOT MB_SEPR_ALR_4;
MB_SEPR_RUN_4 := SEPR_RUN_4;
(* Network 12 *)
OIL_ST_RUN_3 := NOT MILL_ALR_STOP_3 AND (MILL_AUTO_3 AND SEPR_RUN_3 AND SEPR_KM_3 OR MILL_MAN_3) AND (OIL_ST_START_3 OR OIL_ST_RUN_3) AND OIL_ST_STOP_3 AND NOT MB_OIL_ST_ALR_3;
MB_OIL_ST_RUN_3 := OIL_ST_RUN_3;
(* Network 13 *)
OIL_ST_RUN_4 := NOT MILL_ALR_STOP_4 AND (MILL_AUTO_4 AND SEPR_RUN_4 AND SEPR_KM_4 OR MILL_MAN_4) AND (OIL_ST_START_4 OR OIL_ST_RUN_4) AND OIL_ST_STOP_4 AND NOT MB_OIL_ST_ALR_4;
MB_OIL_ST_RUN_4 := OIL_ST_RUN_4;
(* Network 14 *)
_p6 := NOT MILL_ALR_STOP_3 AND (MILL_AUTO_3 AND OIL_ST_KM_3 AND SEPR_RUN_3 AND SEPR_KM_3 OR MILL_MAN_3);
IND_MILL_3(START := _p6 AND MILL_RUN_3, kirish := MILL_ENC_3, vaqtIndukt := vaqtInduc);
MB_MILL_ENC_ALR_3 := IND_MILL_3.ALARM;
MILL_RUN_3 := (_p6 AND MILL_START_3 OR IND_MILL_3.OUT) AND MILL_STOP_3 AND NOT MB_MILL_ALR_3;
MB_MILL_RUN_3 := MILL_RUN_3;
(* Network 15 *)
_p7 := NOT MILL_ALR_STOP_4 AND (MILL_AUTO_4 AND OIL_ST_KM_4 AND SEPR_RUN_4 AND SEPR_KM_4 OR MILL_MAN_4);
IND_MILL_4(START := _p7 AND MILL_RUN_4, kirish := MILL_ENC_4, vaqtIndukt := vaqtInduc);
MB_MILL_ENC_ALR_4 := IND_MILL_4.ALARM;
MILL_RUN_4 := (_p7 AND MILL_START_4 OR IND_MILL_4.OUT) AND MILL_STOP_4 AND NOT MB_MILL_ALR_4;
MB_MILL_RUN_4 := MILL_RUN_4;
(* Network 16 *)
FAN_RUN_3 := NOT MILL_ALR_STOP_3 AND (MILL_AUTO_3 AND MILL_RUN_3 AND MILL_KM_3 OR MILL_MAN_3) AND (FAN_START_3 OR FAN_RUN_3) AND FAN_STOP_3 AND NOT MB_FAN_ALR_3;
MB_FAN_RUN_3 := FAN_RUN_3;
(* Network 17 *)
FAN_RUN_4 := NOT MILL_ALR_STOP_4 AND (MILL_AUTO_4 AND MILL_RUN_4 AND MILL_KM_4 OR MILL_MAN_4) AND (FAN_START_4 OR FAN_RUN_4) AND FAN_STOP_4 AND NOT MB_FAN_ALR_4;
MB_FAN_RUN_4 := FAN_RUN_4;
(* Network 18 *)
MAH_YET3 := NOT MILL_ALR_STOP_3 AND (MILL_AUTO_3 AND FAN_KM_3 AND MILL_KM_3 OR MILL_MAN_3) AND (CONV_START_3 OR MAH_YET3) AND CONV_STOP_3;
(* Network 19 *)
MAH_YET4 := NOT MILL_ALR_STOP_4 AND (MILL_AUTO_4 AND FAN_KM_4 AND MILL_KM_4 OR MILL_MAN_4) AND (CONV_START_4 OR MAH_YET4) AND CONV_STOP_4;
(* Network 20 *)
CONV_RUN_3 := NOT MILL_ALR_STOP_3 AND MAH_YET3 AND MATER_FULL_3 AND NOT MB_CONV_ALR_3;
MB_CONV_RUN_3 := CONV_RUN_3;
(* Network 21 *)
CONV_RUN_4 := NOT MILL_ALR_STOP_4 AND MAH_YET4 AND MATER_FULL_4 AND NOT MB_CONV_ALR_4;
MB_CONV_RUN_4 := CONV_RUN_4;
(* Network 22 *)
VIBRATOR3_T := NOT MILL_ALR_STOP_3 AND (MILL_AUTO_3 OR MILL_MAN_3) AND (VIBR_START_3 OR VIBRATOR3_T) AND VIBR_STOP_3;
(* Network 23 *)
VIBRATOR4_T := NOT MILL_ALR_STOP_4 AND (MILL_AUTO_4 OR MILL_MAN_4) AND (VIBR_START_4 OR VIBRATOR4_T) AND VIBR_STOP_4;
(* Network 24 *)
VALV_RUN_3 := NOT MILL_ALR_STOP_3 AND (MILL_AUTO_3 OR MILL_MAN_3) AND SEPR_KM_3 AND SEPR_RUN_3;
MB_VALV_RUN_3 := VALV_RUN_3;
(* Network 25 *)
VALV_RUN_4 := NOT MILL_ALR_STOP_4 AND (MILL_AUTO_4 OR MILL_MAN_4) AND SEPR_KM_4 AND SEPR_RUN_4;
MB_VALV_RUN_4 := VALV_RUN_4;
(* Network 26 *)
TON1(IN := NOT TON2.Q, PT := VAQT1);
VIBR_RUN_3 := TON1.Q AND VIBRATOR3_T AND CONV_KM_3 AND NOT MB_VIBR_ALR_3;
MB_VIBR_RUN_3 := VIBR_RUN_3;
(* Network 27 *)
TON1(IN := NOT TON2.Q, PT := VAQT2);
VIBR_RUN_4 := TON1.Q AND VIBRATOR4_T AND CONV_KM_4 AND NOT MB_VIBR_ALR_4;
MB_VIBR_RUN_4 := VIBR_RUN_4;
(* Network 28 *)
TON2(IN := TON1.Q, PT := VAQT);
END_PROGRAM

(* POU INDUKTIV, CFC *)
FUNCTION_BLOCK INDUKTIV
VAR_IN_OUT

	(*RESET : BOOL;*)

END_VAR
VAR_INPUT
	START : BOOL;
	kirish : BOOL;
	vaqtIndukt : WORD := 15;
END_VAR

VAR_OUTPUT

	OUT : BOOL;
	ALARM : BOOL;
END_VAR
VAR
	ton1: TON;
	vaqt : TIME;
	ton2: TON;
	TP1: TP;
	TP2: TP;


END_VAR
VAR (* helpers for the ST form of the networks *)
	_t11 : BOOL;
	_t41 : BOOL;
	_t47 : BOOL;
END_VAR
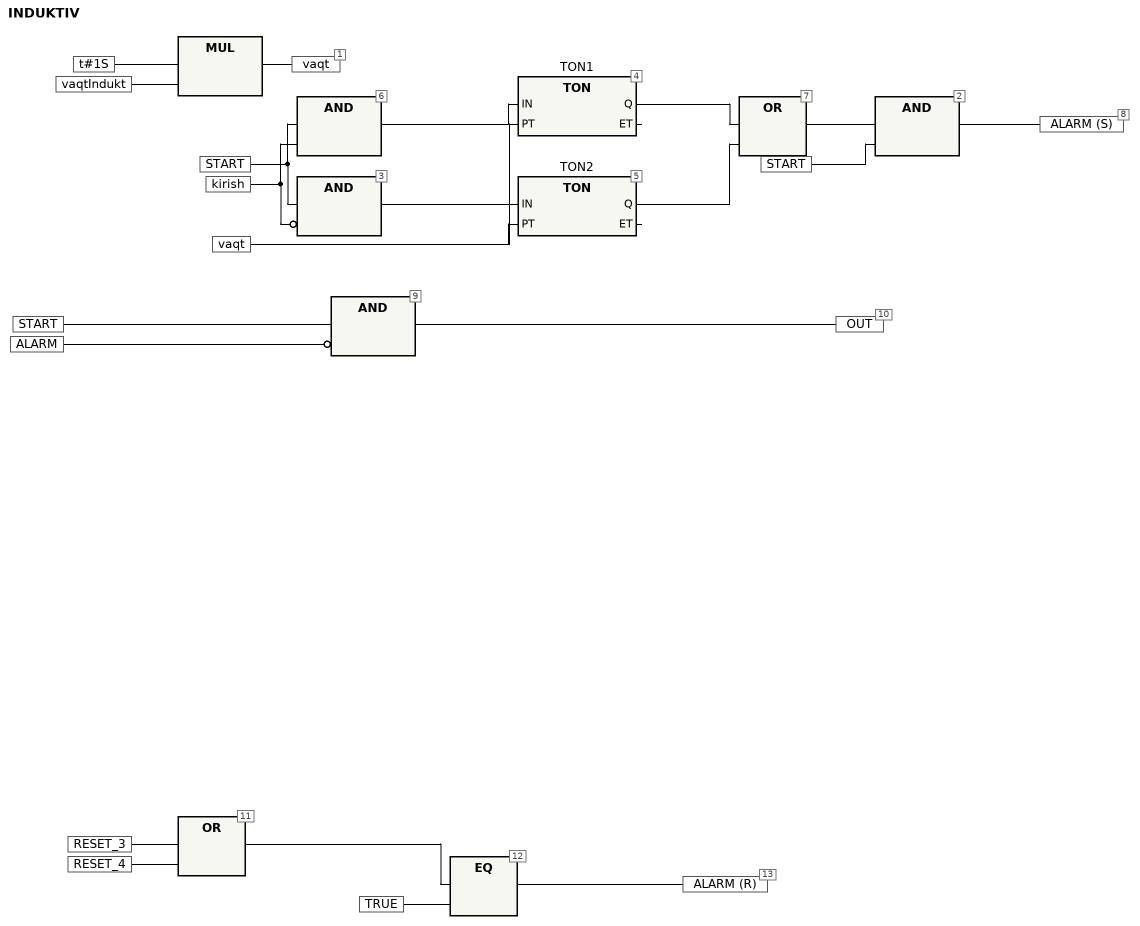
_CFC_ (* Continuous Function Chart, elements in execution order *)
#0 MUL(t#1S, vaqtIndukt)
#1 vaqt <= #0
#2 AND(#7, START)
#3 AND(START, NOT kirish)
#4 TON1:TON(IN: #6, PT: vaqt)
#5 TON2:TON(IN: #3, PT: vaqt)
#6 AND(START, kirish)
#7 OR(#4.Q, #5.Q)
#8 S ALARM <= #2
#9 AND(START, NOT ALARM)
#10 OUT <= #9
#11 OR(RESET_3, RESET_4)
#12 EQ(#11, TRUE)
#13 R ALARM <= #12
_END_CFC_
(* the same logic as Structured Text *)
vaqt := t#1S * vaqtIndukt;
_t41 := _t11 AND START;
TON1(IN := _t47, PT := vaqt);
TON2(IN := START AND NOT kirish, PT := vaqt);
_t47 := START AND kirish;
_t11 := TON1.Q OR TON2.Q;
IF _t41 THEN ALARM := TRUE; END_IF;
OUT := START AND NOT ALARM;
IF (RESET_3 OR RESET_4) = TRUE THEN ALARM := FALSE; END_IF;
END_FUNCTION_BLOCK

(* POU ALARMS, LD *)
PROGRAM ALARMS
VAR
	tofELV: TON;
	tofSHNK3: TON;
	tofSHNK4: TON;
	tofSHNK_SKL_3: TON;
	tofSHNK_SKL_4: TON;
	tofSTAR_31: TON;
	tofSTAR_32: TON;
	tofSTAR_41: TON;
	tofSTAR_42: TON;
	tofSEPR_3: TON;
	tofSEPR_4: TON;
	tofOIL_3: TON;
	tofOIL_4: TON;
	tofMILL_3: TON;
	tofMILL_4: TON;
	tofFAN_3: TON;
	tofFAN_4: TON;
	tofCONV_3: TON;
	tofCONV_4: TON;
	tofVIB_3: TON;
	tofVIB_4: TON;

	vaqt : TIME := T#30S;
END_VAR
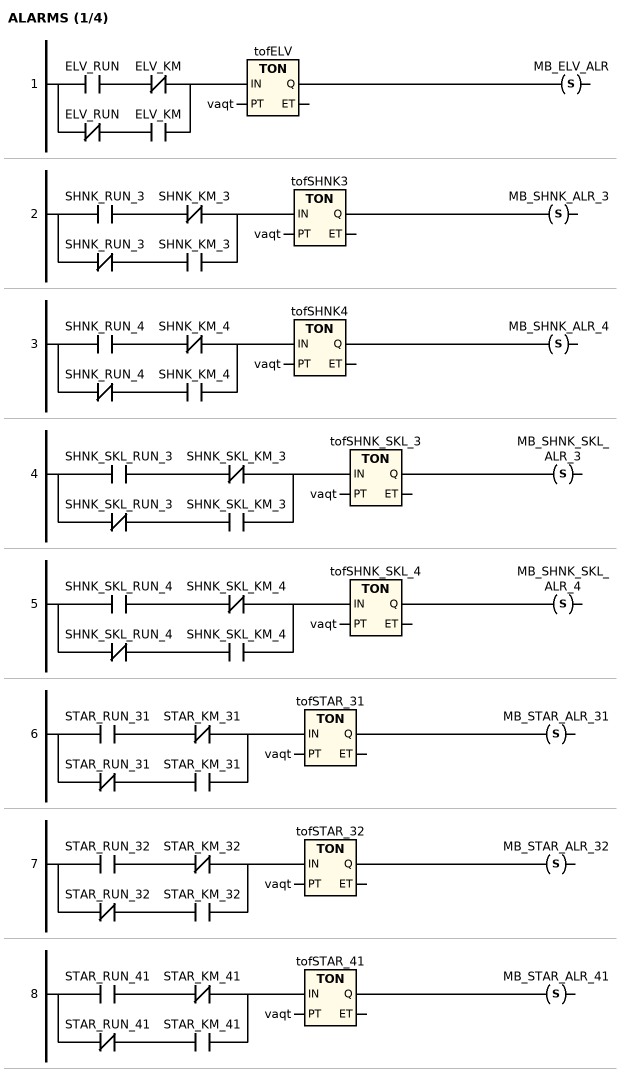
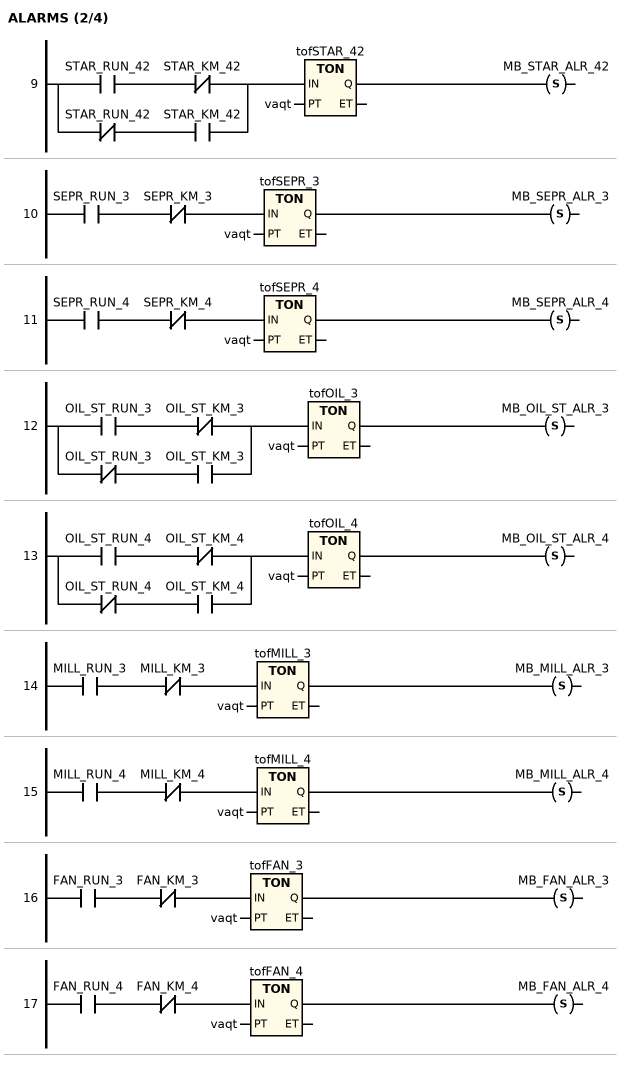
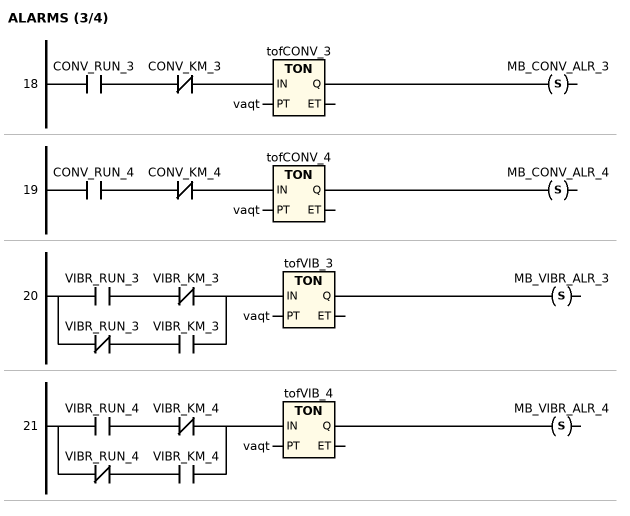
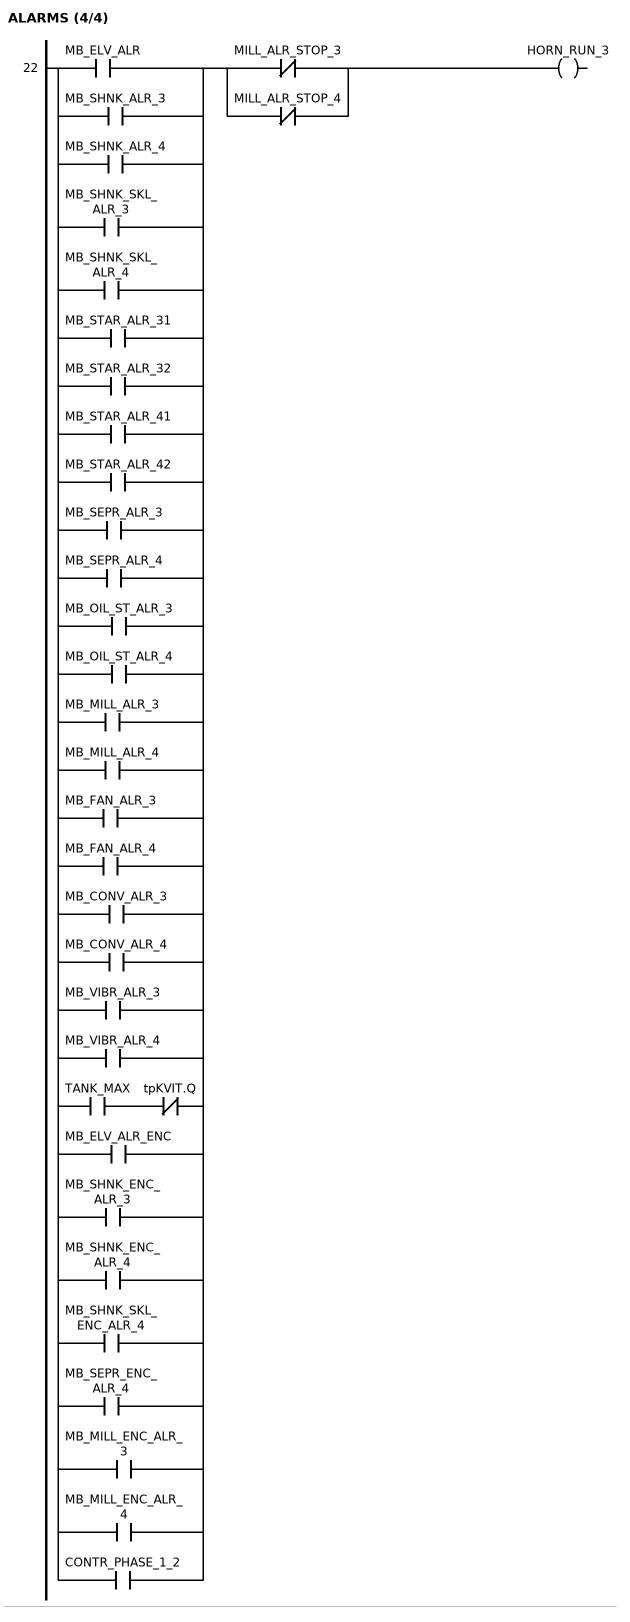
_LD_ (* Ladder Diagram *)
NETWORK 1
	{ [ELV_RUN] - [/ELV_KM] | [/ELV_RUN] - [ELV_KM] } - tofELV:TON(IN: *, PT: vaqt) --- (S MB_ELV_ALR)
NETWORK 2
	{ [SHNK_RUN_3] - [/SHNK_KM_3] | [/SHNK_RUN_3] - [SHNK_KM_3] } - tofSHNK3:TON(IN: *, PT: vaqt) --- (S MB_SHNK_ALR_3)
NETWORK 3
	{ [SHNK_RUN_4] - [/SHNK_KM_4] | [/SHNK_RUN_4] - [SHNK_KM_4] } - tofSHNK4:TON(IN: *, PT: vaqt) --- (S MB_SHNK_ALR_4)
NETWORK 4
	{ [SHNK_SKL_RUN_3] - [/SHNK_SKL_KM_3] | [/SHNK_SKL_RUN_3] - [SHNK_SKL_KM_3] } - tofSHNK_SKL_3:TON(IN: *, PT: vaqt) --- (S MB_SHNK_SKL_ALR_3)
NETWORK 5
	{ [SHNK_SKL_RUN_4] - [/SHNK_SKL_KM_4] | [/SHNK_SKL_RUN_4] - [SHNK_SKL_KM_4] } - tofSHNK_SKL_4:TON(IN: *, PT: vaqt) --- (S MB_SHNK_SKL_ALR_4)
NETWORK 6
	{ [STAR_RUN_31] - [/STAR_KM_31] | [/STAR_RUN_31] - [STAR_KM_31] } - tofSTAR_31:TON(IN: *, PT: vaqt) --- (S MB_STAR_ALR_31)
NETWORK 7
	{ [STAR_RUN_32] - [/STAR_KM_32] | [/STAR_RUN_32] - [STAR_KM_32] } - tofSTAR_32:TON(IN: *, PT: vaqt) --- (S MB_STAR_ALR_32)
NETWORK 8
	{ [STAR_RUN_41] - [/STAR_KM_41] | [/STAR_RUN_41] - [STAR_KM_41] } - tofSTAR_41:TON(IN: *, PT: vaqt) --- (S MB_STAR_ALR_41)
NETWORK 9
	{ [STAR_RUN_42] - [/STAR_KM_42] | [/STAR_RUN_42] - [STAR_KM_42] } - tofSTAR_42:TON(IN: *, PT: vaqt) --- (S MB_STAR_ALR_42)
NETWORK 10
	[SEPR_RUN_3] - [/SEPR_KM_3] - tofSEPR_3:TON(IN: *, PT: vaqt) --- (S MB_SEPR_ALR_3)
NETWORK 11
	[SEPR_RUN_4] - [/SEPR_KM_4] - tofSEPR_4:TON(IN: *, PT: vaqt) --- (S MB_SEPR_ALR_4)
NETWORK 12
	{ [OIL_ST_RUN_3] - [/OIL_ST_KM_3] | [/OIL_ST_RUN_3] - [OIL_ST_KM_3] } - tofOIL_3:TON(IN: *, PT: vaqt) --- (S MB_OIL_ST_ALR_3)
NETWORK 13
	{ [OIL_ST_RUN_4] - [/OIL_ST_KM_4] | [/OIL_ST_RUN_4] - [OIL_ST_KM_4] } - tofOIL_4:TON(IN: *, PT: vaqt) --- (S MB_OIL_ST_ALR_4)
NETWORK 14
	[MILL_RUN_3] - [/MILL_KM_3] - tofMILL_3:TON(IN: *, PT: vaqt) --- (S MB_MILL_ALR_3)
NETWORK 15
	[MILL_RUN_4] - [/MILL_KM_4] - tofMILL_4:TON(IN: *, PT: vaqt) --- (S MB_MILL_ALR_4)
NETWORK 16
	[FAN_RUN_3] - [/FAN_KM_3] - tofFAN_3:TON(IN: *, PT: vaqt) --- (S MB_FAN_ALR_3)
NETWORK 17
	[FAN_RUN_4] - [/FAN_KM_4] - tofFAN_4:TON(IN: *, PT: vaqt) --- (S MB_FAN_ALR_4)
NETWORK 18
	[CONV_RUN_3] - [/CONV_KM_3] - tofCONV_3:TON(IN: *, PT: vaqt) --- (S MB_CONV_ALR_3)
NETWORK 19
	[CONV_RUN_4] - [/CONV_KM_4] - tofCONV_4:TON(IN: *, PT: vaqt) --- (S MB_CONV_ALR_4)
NETWORK 20
	{ [VIBR_RUN_3] - [/VIBR_KM_3] | [/VIBR_RUN_3] - [VIBR_KM_3] } - tofVIB_3:TON(IN: *, PT: vaqt) --- (S MB_VIBR_ALR_3)
NETWORK 21
	{ [VIBR_RUN_4] - [/VIBR_KM_4] | [/VIBR_RUN_4] - [VIBR_KM_4] } - tofVIB_4:TON(IN: *, PT: vaqt) --- (S MB_VIBR_ALR_4)
NETWORK 22
	{ [MB_ELV_ALR] | [MB_SHNK_ALR_3] | [MB_SHNK_ALR_4] | [MB_SHNK_SKL_ALR_3] | [MB_SHNK_SKL_ALR_4] | [MB_STAR_ALR_31] | [MB_STAR_ALR_32] | [MB_STAR_ALR_41] | [MB_STAR_ALR_42] | [MB_SEPR_ALR_3] | [MB_SEPR_ALR_4] | [MB_OIL_ST_ALR_3] | [MB_OIL_ST_ALR_4] | [MB_MILL_ALR_3] | [MB_MILL_ALR_4] | [MB_FAN_ALR_3] | [MB_FAN_ALR_4] | [MB_CONV_ALR_3] | [MB_CONV_ALR_4] | [MB_VIBR_ALR_3] | [MB_VIBR_ALR_4] | [TANK_MAX] - [/tpKVIT.Q] | [MB_ELV_ALR_ENC] | [MB_SHNK_ENC_ALR_3] | [MB_SHNK_ENC_ALR_4] | [MB_SHNK_SKL_ENC_ALR_4] | [MB_SEPR_ENC_ALR_4] | [MB_MILL_ENC_ALR_3] | [MB_MILL_ENC_ALR_4] | [CONTR_PHASE_1_2] } - { [/MILL_ALR_STOP_3] | [/MILL_ALR_STOP_4] } --- (HORN_RUN_3)
_END_LD_
(* the same logic as Structured Text *)
(* Network 1 *)
tofELV(IN := ELV_RUN AND NOT ELV_KM OR NOT ELV_RUN AND ELV_KM, PT := vaqt);
IF tofELV.Q THEN MB_ELV_ALR := TRUE; END_IF;
(* Network 2 *)
tofSHNK3(IN := SHNK_RUN_3 AND NOT SHNK_KM_3 OR NOT SHNK_RUN_3 AND SHNK_KM_3, PT := vaqt);
IF tofSHNK3.Q THEN MB_SHNK_ALR_3 := TRUE; END_IF;
(* Network 3 *)
tofSHNK4(IN := SHNK_RUN_4 AND NOT SHNK_KM_4 OR NOT SHNK_RUN_4 AND SHNK_KM_4, PT := vaqt);
IF tofSHNK4.Q THEN MB_SHNK_ALR_4 := TRUE; END_IF;
(* Network 4 *)
tofSHNK_SKL_3(IN := SHNK_SKL_RUN_3 AND NOT SHNK_SKL_KM_3 OR NOT SHNK_SKL_RUN_3 AND SHNK_SKL_KM_3, PT := vaqt);
IF tofSHNK_SKL_3.Q THEN MB_SHNK_SKL_ALR_3 := TRUE; END_IF;
(* Network 5 *)
tofSHNK_SKL_4(IN := SHNK_SKL_RUN_4 AND NOT SHNK_SKL_KM_4 OR NOT SHNK_SKL_RUN_4 AND SHNK_SKL_KM_4, PT := vaqt);
IF tofSHNK_SKL_4.Q THEN MB_SHNK_SKL_ALR_4 := TRUE; END_IF;
(* Network 6 *)
tofSTAR_31(IN := STAR_RUN_31 AND NOT STAR_KM_31 OR NOT STAR_RUN_31 AND STAR_KM_31, PT := vaqt);
IF tofSTAR_31.Q THEN MB_STAR_ALR_31 := TRUE; END_IF;
(* Network 7 *)
tofSTAR_32(IN := STAR_RUN_32 AND NOT STAR_KM_32 OR NOT STAR_RUN_32 AND STAR_KM_32, PT := vaqt);
IF tofSTAR_32.Q THEN MB_STAR_ALR_32 := TRUE; END_IF;
(* Network 8 *)
tofSTAR_41(IN := STAR_RUN_41 AND NOT STAR_KM_41 OR NOT STAR_RUN_41 AND STAR_KM_41, PT := vaqt);
IF tofSTAR_41.Q THEN MB_STAR_ALR_41 := TRUE; END_IF;
(* Network 9 *)
tofSTAR_42(IN := STAR_RUN_42 AND NOT STAR_KM_42 OR NOT STAR_RUN_42 AND STAR_KM_42, PT := vaqt);
IF tofSTAR_42.Q THEN MB_STAR_ALR_42 := TRUE; END_IF;
(* Network 10 *)
tofSEPR_3(IN := SEPR_RUN_3 AND NOT SEPR_KM_3, PT := vaqt);
IF tofSEPR_3.Q THEN MB_SEPR_ALR_3 := TRUE; END_IF;
(* Network 11 *)
tofSEPR_4(IN := SEPR_RUN_4 AND NOT SEPR_KM_4, PT := vaqt);
IF tofSEPR_4.Q THEN MB_SEPR_ALR_4 := TRUE; END_IF;
(* Network 12 *)
tofOIL_3(IN := OIL_ST_RUN_3 AND NOT OIL_ST_KM_3 OR NOT OIL_ST_RUN_3 AND OIL_ST_KM_3, PT := vaqt);
IF tofOIL_3.Q THEN MB_OIL_ST_ALR_3 := TRUE; END_IF;
(* Network 13 *)
tofOIL_4(IN := OIL_ST_RUN_4 AND NOT OIL_ST_KM_4 OR NOT OIL_ST_RUN_4 AND OIL_ST_KM_4, PT := vaqt);
IF tofOIL_4.Q THEN MB_OIL_ST_ALR_4 := TRUE; END_IF;
(* Network 14 *)
tofMILL_3(IN := MILL_RUN_3 AND NOT MILL_KM_3, PT := vaqt);
IF tofMILL_3.Q THEN MB_MILL_ALR_3 := TRUE; END_IF;
(* Network 15 *)
tofMILL_4(IN := MILL_RUN_4 AND NOT MILL_KM_4, PT := vaqt);
IF tofMILL_4.Q THEN MB_MILL_ALR_4 := TRUE; END_IF;
(* Network 16 *)
tofFAN_3(IN := FAN_RUN_3 AND NOT FAN_KM_3, PT := vaqt);
IF tofFAN_3.Q THEN MB_FAN_ALR_3 := TRUE; END_IF;
(* Network 17 *)
tofFAN_4(IN := FAN_RUN_4 AND NOT FAN_KM_4, PT := vaqt);
IF tofFAN_4.Q THEN MB_FAN_ALR_4 := TRUE; END_IF;
(* Network 18 *)
tofCONV_3(IN := CONV_RUN_3 AND NOT CONV_KM_3, PT := vaqt);
IF tofCONV_3.Q THEN MB_CONV_ALR_3 := TRUE; END_IF;
(* Network 19 *)
tofCONV_4(IN := CONV_RUN_4 AND NOT CONV_KM_4, PT := vaqt);
IF tofCONV_4.Q THEN MB_CONV_ALR_4 := TRUE; END_IF;
(* Network 20 *)
tofVIB_3(IN := VIBR_RUN_3 AND NOT VIBR_KM_3 OR NOT VIBR_RUN_3 AND VIBR_KM_3, PT := vaqt);
IF tofVIB_3.Q THEN MB_VIBR_ALR_3 := TRUE; END_IF;
(* Network 21 *)
tofVIB_4(IN := VIBR_RUN_4 AND NOT VIBR_KM_4 OR NOT VIBR_RUN_4 AND VIBR_KM_4, PT := vaqt);
IF tofVIB_4.Q THEN MB_VIBR_ALR_4 := TRUE; END_IF;
(* Network 22 *)
HORN_RUN_3 := (MB_ELV_ALR OR MB_SHNK_ALR_3 OR MB_SHNK_ALR_4 OR MB_SHNK_SKL_ALR_3 OR MB_SHNK_SKL_ALR_4 OR MB_STAR_ALR_31 OR MB_STAR_ALR_32 OR MB_STAR_ALR_41 OR MB_STAR_ALR_42 OR MB_SEPR_ALR_3 OR MB_SEPR_ALR_4 OR MB_OIL_ST_ALR_3 OR MB_OIL_ST_ALR_4 OR MB_MILL_ALR_3 OR MB_MILL_ALR_4 OR MB_FAN_ALR_3 OR MB_FAN_ALR_4 OR MB_CONV_ALR_3 OR MB_CONV_ALR_4 OR MB_VIBR_ALR_3 OR MB_VIBR_ALR_4 OR TANK_MAX AND NOT tpKVIT.Q OR MB_ELV_ALR_ENC OR MB_SHNK_ENC_ALR_3 OR MB_SHNK_ENC_ALR_4 OR MB_SHNK_SKL_ENC_ALR_4 OR MB_SEPR_ENC_ALR_4 OR MB_MILL_ENC_ALR_3 OR MB_MILL_ENC_ALR_4 OR CONTR_PHASE_1_2) AND (NOT MILL_ALR_STOP_3 OR NOT MILL_ALR_STOP_4);
END_PROGRAM

(* POU RESET_ALRM, LD *)
PROGRAM RESET_ALRM
VAR
END_VAR
VAR (* helpers for the ST form of the networks *)
	_p1 : BOOL;
END_VAR
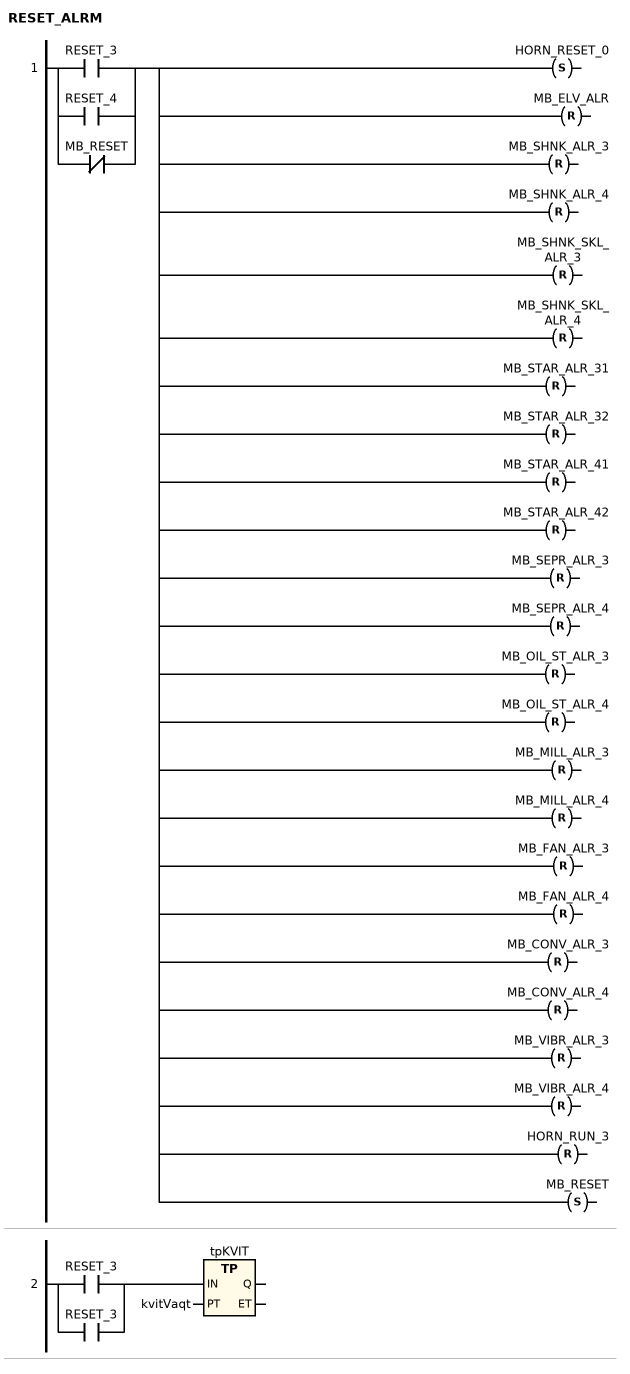
_LD_ (* Ladder Diagram *)
NETWORK 1
	{ [RESET_3] | [RESET_4] | [/MB_RESET] } --- (S HORN_RESET_0) (R MB_ELV_ALR) (R MB_SHNK_ALR_3) (R MB_SHNK_ALR_4) (R MB_SHNK_SKL_ALR_3) (R MB_SHNK_SKL_ALR_4) (R MB_STAR_ALR_31) (R MB_STAR_ALR_32) (R MB_STAR_ALR_41) (R MB_STAR_ALR_42) (R MB_SEPR_ALR_3) (R MB_SEPR_ALR_4) (R MB_OIL_ST_ALR_3) (R MB_OIL_ST_ALR_4) (R MB_MILL_ALR_3) (R MB_MILL_ALR_4) (R MB_FAN_ALR_3) (R MB_FAN_ALR_4) (R MB_CONV_ALR_3) (R MB_CONV_ALR_4) (R MB_VIBR_ALR_3) (R MB_VIBR_ALR_4) (R HORN_RUN_3) (S MB_RESET)
NETWORK 2
	{ [RESET_3] | [RESET_3] } - tpKVIT:TP(IN: *, PT: kvitVaqt)
_END_LD_
(* the same logic as Structured Text *)
(* Network 1 *)
_p1 := RESET_3 OR RESET_4 OR NOT MB_RESET;
IF _p1 THEN HORN_RESET_0 := TRUE; MB_ELV_ALR := FALSE; MB_SHNK_ALR_3 := FALSE; MB_SHNK_ALR_4 := FALSE; MB_SHNK_SKL_ALR_3 := FALSE; MB_SHNK_SKL_ALR_4 := FALSE; MB_STAR_ALR_31 := FALSE; MB_STAR_ALR_32 := FALSE; MB_STAR_ALR_41 := FALSE; MB_STAR_ALR_42 := FALSE; MB_SEPR_ALR_3 := FALSE; MB_SEPR_ALR_4 := FALSE; MB_OIL_ST_ALR_3 := FALSE; MB_OIL_ST_ALR_4 := FALSE; MB_MILL_ALR_3 := FALSE; MB_MILL_ALR_4 := FALSE; MB_FAN_ALR_3 := FALSE; MB_FAN_ALR_4 := FALSE; MB_CONV_ALR_3 := FALSE; MB_CONV_ALR_4 := FALSE; MB_VIBR_ALR_3 := FALSE; MB_VIBR_ALR_4 := FALSE; HORN_RUN_3 := FALSE; MB_RESET := TRUE; END_IF;
(* Network 2 *)
tpKVIT(IN := RESET_3 OR RESET_3, PT := kvitVaqt);
END_PROGRAM

(* POU TRANSLATE, ST *)
PROGRAM TRANSLATE
VAR
	CON1: LIN_TRAFO;
	CON2: LIN_TRAFO;
	CON3: LIN_TRAFO;
	CON4: LIN_TRAFO;
	CON5: LIN_TRAFO;
	CON6: LIN_TRAFO;
	CON7: LIN_TRAFO;
	CON8: LIN_TRAFO;
	IN_MIN : REAL := 4;
	IN_MAX: REAL := 20;
	OUT_MIN_SEN : REAL := -10;
	OUT_MAX_SEN: REAL := 1;
	OUT_MIN_CUR : REAL := 0;
	OUT_MAX_CUR: REAL := 50;
END_VAR
MB_ANALOG();

MV8();
MV16();
MV24();
MU32_OUT();
MV48();
MB_TANK_MIN := TANK_MIN;
MB_TANK_MIDLE := TANK_MIDL;
MB_TANK_MAX := TANK_MAX;
END_PROGRAM
ACTION MB_ANALOG:
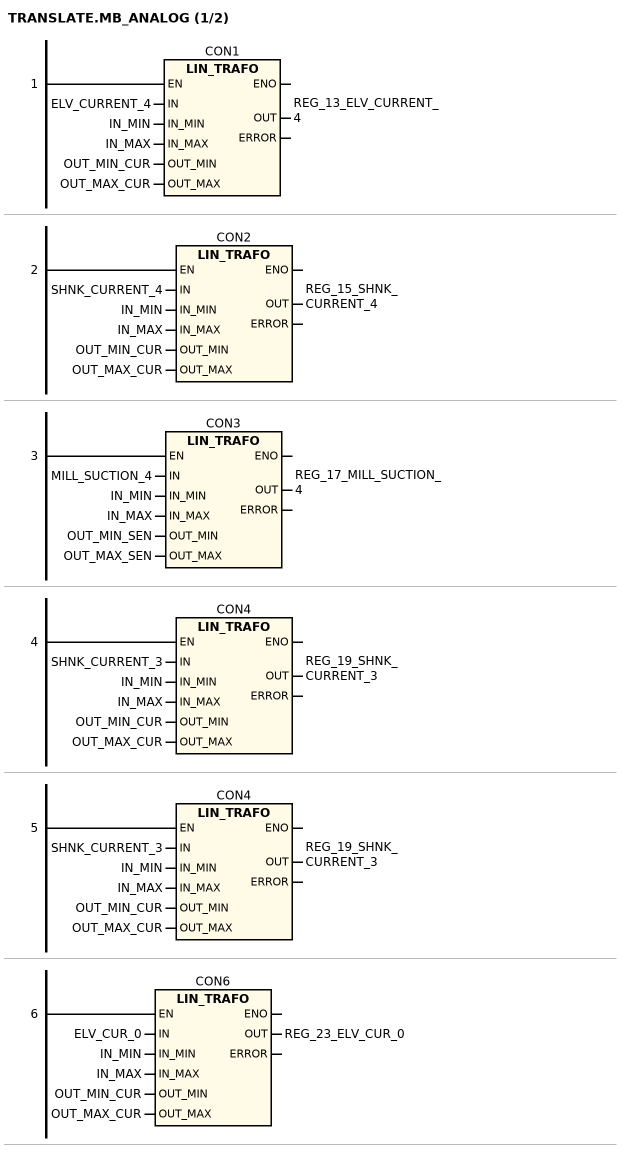
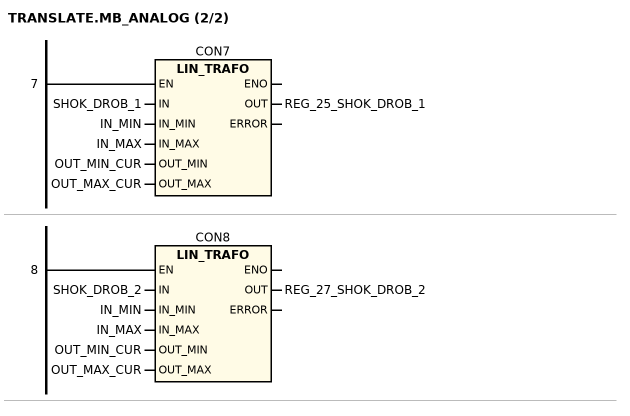
_LD_ (* Ladder Diagram *)
NETWORK 1
	*
		EN --- CON1:LIN_TRAFO(IN: ELV_CURRENT_4, IN_MIN: IN_MIN, IN_MAX: IN_MAX, OUT_MIN: OUT_MIN_CUR, OUT_MAX: OUT_MAX_CUR) => REG_13_ELV_CURRENT_4
NETWORK 2
	*
		EN --- CON2:LIN_TRAFO(IN: SHNK_CURRENT_4, IN_MIN: IN_MIN, IN_MAX: IN_MAX, OUT_MIN: OUT_MIN_CUR, OUT_MAX: OUT_MAX_CUR) => REG_15_SHNK_CURRENT_4
NETWORK 3
	*
		EN --- CON3:LIN_TRAFO(IN: MILL_SUCTION_4, IN_MIN: IN_MIN, IN_MAX: IN_MAX, OUT_MIN: OUT_MIN_SEN, OUT_MAX: OUT_MAX_SEN) => REG_17_MILL_SUCTION_4
NETWORK 4
	*
		EN --- CON4:LIN_TRAFO(IN: SHNK_CURRENT_3, IN_MIN: IN_MIN, IN_MAX: IN_MAX, OUT_MIN: OUT_MIN_CUR, OUT_MAX: OUT_MAX_CUR) => REG_19_SHNK_CURRENT_3
NETWORK 5
	*
		EN --- CON4:LIN_TRAFO(IN: SHNK_CURRENT_3, IN_MIN: IN_MIN, IN_MAX: IN_MAX, OUT_MIN: OUT_MIN_CUR, OUT_MAX: OUT_MAX_CUR) => REG_19_SHNK_CURRENT_3
NETWORK 6
	*
		EN --- CON6:LIN_TRAFO(IN: ELV_CUR_0, IN_MIN: IN_MIN, IN_MAX: IN_MAX, OUT_MIN: OUT_MIN_CUR, OUT_MAX: OUT_MAX_CUR) => REG_23_ELV_CUR_0
NETWORK 7
	*
		EN --- CON7:LIN_TRAFO(IN: SHOK_DROB_1, IN_MIN: IN_MIN, IN_MAX: IN_MAX, OUT_MIN: OUT_MIN_CUR, OUT_MAX: OUT_MAX_CUR) => REG_25_SHOK_DROB_1
NETWORK 8
	*
		EN --- CON8:LIN_TRAFO(IN: SHOK_DROB_2, IN_MIN: IN_MIN, IN_MAX: IN_MAX, OUT_MIN: OUT_MIN_CUR, OUT_MAX: OUT_MAX_CUR) => REG_27_SHOK_DROB_2
_END_LD_
(* the same logic as Structured Text *)
(* Network 1 *)
CON1(IN := ELV_CURRENT_4, IN_MIN := IN_MIN, IN_MAX := IN_MAX, OUT_MIN := OUT_MIN_CUR, OUT_MAX := OUT_MAX_CUR);
REG_13_ELV_CURRENT_4 := CON1.OUT;
(* Network 2 *)
CON2(IN := SHNK_CURRENT_4, IN_MIN := IN_MIN, IN_MAX := IN_MAX, OUT_MIN := OUT_MIN_CUR, OUT_MAX := OUT_MAX_CUR);
REG_15_SHNK_CURRENT_4 := CON2.OUT;
(* Network 3 *)
CON3(IN := MILL_SUCTION_4, IN_MIN := IN_MIN, IN_MAX := IN_MAX, OUT_MIN := OUT_MIN_SEN, OUT_MAX := OUT_MAX_SEN);
REG_17_MILL_SUCTION_4 := CON3.OUT;
(* Network 4 *)
CON4(IN := SHNK_CURRENT_3, IN_MIN := IN_MIN, IN_MAX := IN_MAX, OUT_MIN := OUT_MIN_CUR, OUT_MAX := OUT_MAX_CUR);
REG_19_SHNK_CURRENT_3 := CON4.OUT;
(* Network 5 *)
CON4(IN := SHNK_CURRENT_3, IN_MIN := IN_MIN, IN_MAX := IN_MAX, OUT_MIN := OUT_MIN_CUR, OUT_MAX := OUT_MAX_CUR);
REG_19_SHNK_CURRENT_3 := CON4.OUT;
(* Network 6 *)
CON6(IN := ELV_CUR_0, IN_MIN := IN_MIN, IN_MAX := IN_MAX, OUT_MIN := OUT_MIN_CUR, OUT_MAX := OUT_MAX_CUR);
REG_23_ELV_CUR_0 := CON6.OUT;
(* Network 7 *)
CON7(IN := SHOK_DROB_1, IN_MIN := IN_MIN, IN_MAX := IN_MAX, OUT_MIN := OUT_MIN_CUR, OUT_MAX := OUT_MAX_CUR);
REG_25_SHOK_DROB_1 := CON7.OUT;
(* Network 8 *)
CON8(IN := SHOK_DROB_2, IN_MIN := IN_MIN, IN_MAX := IN_MAX, OUT_MIN := OUT_MIN_CUR, OUT_MAX := OUT_MAX_CUR);
REG_27_SHOK_DROB_2 := CON8.OUT;
END_ACTION
ACTION MU32_OUT:
MU01 := BOOL_TO_WORD(ELV_RUN) * 1000;
MU02 := BOOL_TO_WORD(SHNK_RUN_4) * 1000;
MU03 := BOOL_TO_WORD(SHNK_SKL_RUN_4) * 1000;
MU04 := BOOL_TO_WORD(STAR_RUN_41) * 1000;
MU05 := BOOL_TO_WORD(STAR_RUN_42) * 1000;
MU06 := BOOL_TO_WORD(SEPR_RUN_4) * 1000;
MU07 := BOOL_TO_WORD(OIL_ST_RUN_4) * 1000;
MU08 := BOOL_TO_WORD(MILL_RUN_4) * 1000;
MU09 := BOOL_TO_WORD(FAN_RUN_4) * 1000;
MU10 := BOOL_TO_WORD(CONV_RUN_4) * 1000;
MU11 := BOOL_TO_WORD(VIBR_RUN_4) * 1000;
MU12 := BOOL_TO_WORD(VALV_RUN_4) * 1000;
MU13 := BOOL_TO_WORD(HORN_RUN_4) * 1000;
(*
MU14 := BOOL_TO_WORD(m_out14) * 1000;
MU15 := BOOL_TO_WORD(m_out15) * 1000;
MU16 := BOOL_TO_WORD(m_out16) * 1000;
*)
MU17 := BOOL_TO_WORD(ELV_RUN) * 1000;
MU18 := BOOL_TO_WORD(SHNK_RUN_3) * 1000;
MU19 := BOOL_TO_WORD(SHNK_SKL_RUN_3) * 1000;
MU20 := BOOL_TO_WORD(STAR_RUN_31) * 1000;
MU21 := BOOL_TO_WORD(STAR_RUN_32) * 1000;
MU22 := BOOL_TO_WORD(SEPR_RUN_3) * 1000;
MU23 := BOOL_TO_WORD(OIL_ST_RUN_3) * 1000;
MU24 := BOOL_TO_WORD(MILL_RUN_3) * 1000;
MU25 := BOOL_TO_WORD(FAN_RUN_3) * 1000;
MU26 := BOOL_TO_WORD(CONV_RUN_3) * 1000;
MU27 := BOOL_TO_WORD(VIBR_RUN_3) * 1000;
MU28 := BOOL_TO_WORD(VALV_RUN_3) * 1000;
MU29 := BOOL_TO_WORD(HORN_RUN_3) * 1000;
(*
MU30 := BOOL_TO_WORD(m_out30) * 1000;
MU31 := BOOL_TO_WORD(m_out31) * 1000;
MU32 := BOOL_TO_WORD(m_out32) * 1000;
*)
END_ACTION
ACTION MV16:
STAR_STOP_32 := MV16_0.0;
SEPR_STOP_3 := MV16_0.1;
OIL_ST_STOP_3 := MV16_0.2;
MILL_STOP_3 := MV16_0.3;
FAN_STOP_3 := MV16_0.4;
CONV_STOP_3 := MV16_0.5;
VIBR_STOP_3 := MV16_0.6;
(**********************)

STAR_START_32 := MV16_0.8;
SEPR_START_3 := MV16_0.9;
OIL_ST_START_3 := MV16_0.10;
MILL_START_3 := MV16_0.11;
FAN_START_3 := MV16_0.12;
CONV_START_3 := MV16_0.13;
VIBR_START_3 := MV16_0.14;
END_ACTION
ACTION MV24:
ELV_KM := MV24_0.0;
SHNK_KM_4 := MV24_0.1;
SHNK_SKL_KM_4 := MV24_0.2;
STAR_KM_41 := MV24_0.3;
STAR_KM_42 := MV24_0.4;
SEPR_KM_4 := MV24_0.5;
OIL_ST_KM_4 := MV24_0.6;
MILL_KM_4 := MV24_0.7;
MB_MATER_FULL_4 := MATER_FULL_4 := MV24_0.8;
FAN_KM_4 := MV24_0.9;
CONV_KM_4 := MV24_0.10;
VIBR_KM_4 := MV24_0.11;
(*********
ELV_KM_3 := MV24_1.0;*)
SHNK_KM_3 := MV24_1.1;
SHNK_SKL_KM_3 := MV24_1.2;
STAR_KM_31 := MV24_1.3;
STAR_KM_32 := MV24_1.4;
SEPR_KM_3 := MV24_1.5;
OIL_ST_KM_3 := MV24_1.6;
MILL_KM_3 := MV24_1.7;
MB_MATER_FULL_3 := MATER_FULL_3 := MV24_1.8;
FAN_KM_3 := MV24_1.9;
CONV_KM_3 := MV24_1.10;
VIBR_KM_3 := MV24_1.11;
CONTR_PHASE_1_2  := MV24_1.12;
END_ACTION
ACTION MV48:
	MB_EMER_STOP_0 := MV48_0.0;
	MB_MANUAL_ELV_0 := MV48_0.1;
	MB_AUTO_ELV_0 := MV48_0.2;
	MB_RESET_0 := MV48_0.3;
	MB_ELV_STOP_0 := MV48_0.4;
	MB_ELV_START_0 := MV48_0.5;
	MB_SHOK_DROB_STOP_1  := MV48_0.6;
	MB_SHOK_DROB_START_1 := MV48_0.7;
	MB_SHOK_DROB_STOP_2  := MV48_0.8;
	MB_SHOK_DROB_START_2 := MV48_0.9;
	MB_CONV_STOP_0 := MV48_0.10;
	MB_CONV_START_0 := MV48_0.11;
	(****RESERV CONV ***) (*12*)
	(***RESERV CONV****) (*13*)
	MB_ELV_KM_0 := MV48_0.14;
	MB_SHOK_DROB_KM_1 := MV48_0.15;
	MB_SHOK_DROB_KM_2 := MV48_1.0;
	MB_CONV_KM_0 := MV48_1.1;
	(** RESERV KM CONV **)
	MB_TANK_MAX_0 := MV48_1.3;
	MB_TANK_MIDLE_0 := MV48_1.4;
	MB_TANK_MIN_0 := MV48_1.5;
END_ACTION
ACTION MV8:
ELV_STOP_4 := MV8_0.0;
SHNK_STOP_4 := MV8_0.1;
SHNK_SKL_STOP_4 := MV8_0.2;
STAR_STOP_41 := MV8_0.3;
STAR_STOP_42 := MV8_0.4;
SEPR_STOP_4 := MV8_0.5;
OIL_ST_STOP_4 := MV8_0.6;
MILL_STOP_4 := MV8_0.7;
FAN_STOP_4 := MV8_0.8;
CONV_STOP_4 := MV8_0.9;
VIBR_STOP_4 := MV8_0.10;

ELV_STOP_3 := MV8_0.12;
SHNK_STOP_3 := MV8_0.13;
SHNK_SKL_STOP_3 := MV8_0.14;
STAR_STOP_31 := MV8_0.15;

(**********************)
ELV_START_4 := MV8_1.0;
SHNK_START_4 := MV8_1.1;
SHNK_SKL_START_4 := MV8_1.2;
STAR_START_41 := MV8_1.3;
STAR_START_42 := MV8_1.4;
SEPR_START_4 := MV8_1.5;
OIL_ST_START_4 := MV8_1.6;
MILL_START_4 := MV8_1.7;
FAN_START_4 := MV8_1.8;
CONV_START_4 := MV8_1.9;
VIBR_START_4 := MV8_1.10;

ELV_START_3 := MV8_1.12;
SHNK_START_3 := MV8_1.13;
SHNK_SKL_START_3 := MV8_1.14;
STAR_START_31 := MV8_1.15;
END_ACTION
ACTION TR_REG_1:
(*
REG_1.0 := MB_ELV_ALR;
REG_1.1 := MB_ELV_ALR_ENC;
REG_1.2 := MB_SHNK_ALR_4;
REG_1.3 :=MB_SHNK_ENC_ALR_4 ;
REG_1.4 := MB_SHNK_SKL_ALR_4;
REG_1.5 := MB_SHNK_SKL_ENC_ALR_4;
REG_1.6 :=MB_STAR_ALR_41 ;
REG_1.7 := MB_STAR_ALR_42;

REG_1.8 := MB_SEPR_ALR_4;
REG_1.9 := MB_OIL_ST_ALR_4;
REG_1.10 :=MB_MILL_ALR_4 ;
REG_1.11 := MB_FAN_ALR_4;
REG_1.12 := MB_CONV_ALR_4;
REG_1.13 := MB_VIBR_ALR_4 ;
REG_1.14 := MB_MILL_ENC_ALR_4;
REG_1.15 := MB_SEPR_ENC_ALR_4;
*);
END_ACTION
ACTION TR_REG_2:
(*
REG_2.0 := MB_SHNK_ALR_3;
REG_2.1 := MB_SHNK_ENC_ALR_3;
REG_2.2 := MB_SHNK_SKL_ALR_3;
REG_2.3 := MB_STAR_ALR_31;
REG_2.4 := MB_STAR_ALR_32;
REG_2.5 := MB_SEPR_ALR_3;
REG_2.6 := MB_SEPR_ENC_ALR_3;
REG_2.7 := MB_OIL_ST_ALR_3;

REG_2.8 := MB_MILL_ALR_3;
REG_2.10 := MB_FAN_ALR_3;
REG_2.11 := MB_CONV_ALR_3;
REG_2.12 := MB_VIBR_ALR_3;
REG_2.13 := MB_MILL_ENC_ALR_3;
REG_2.14 := MB_TANK_MIN;
REG_2.15 := MB_TANK_MAX;

*)
;
END_ACTION
ACTION TR_REG_3:
(*
REG_3.0 := MB_ELV_RUN;
REG_3.1 := MB_SHNK_RUN_4;
REG_3.2 := MB_SHNK_SKL_RUN_4;
REG_3.3 := MB_STAR_RUN_41;
REG_3.4 := MB_STAR_RUN_42;
REG_3.5 := MB_SEPR_RUN_4;
REG_3.6 := MB_OIL_ST_RUN_4;
REG_3.7 := MB_MILL_RUN_4;

REG_3.8 := MB_FAN_RUN_4;
REG_3.9 := MB_CONV_RUN_4;
REG_3.10 := MB_VIBR_RUN_4;
REG_3.11 := MB_VALV_RUN_4;
REG_3.12 := MB_HORN_RUN;
REG_3.13 := MB_MATER_FULL_4;

*)
;
END_ACTION
ACTION TR_REG_4:
(*
REG_4.0 := MB_SHNK_RUN_3;
REG_4.1 := MB_SHNK_SKL_RUN_3;
REG_4.2 := MB_STAR_RUN_31;
REG_4.3 := MB_STAR_RUN_32;
REG_4.4 := MB_SEPR_RUN_3;
REG_4.5 := MB_OIL_ST_RUN_3;
REG_4.6 := MB_MILL_RUN_3;
REG_4.7 := MB_FAN_RUN_3;

REG_4.8 := MB_CONV_RUN_3;
REG_4.9 := MB_VIBR_RUN_3;
REG_4.10 := MB_VALV_RUN_3;
REG_4.11 := MB_MATER_FULL_3;

*)
;
END_ACTION

(* POU DROBILKA, LD *)
PROGRAM DROBILKA
VAR
	convTON : TON;
	conVAQT : TIME := T#180s;
	drobTON : TON;
	drobVAQT: TIME := T#180s;
	maxTON : TON;
	maxVAQT: TIME := T#5s;
	ELV_F_TRIG: F_TRIG;
	TANK_FULL: BOOL;
	ELV_R_TRIG: R_TRIG;
END_VAR
VAR (* helpers for the ST form of the networks *)
	_p1 : BOOL;
END_VAR
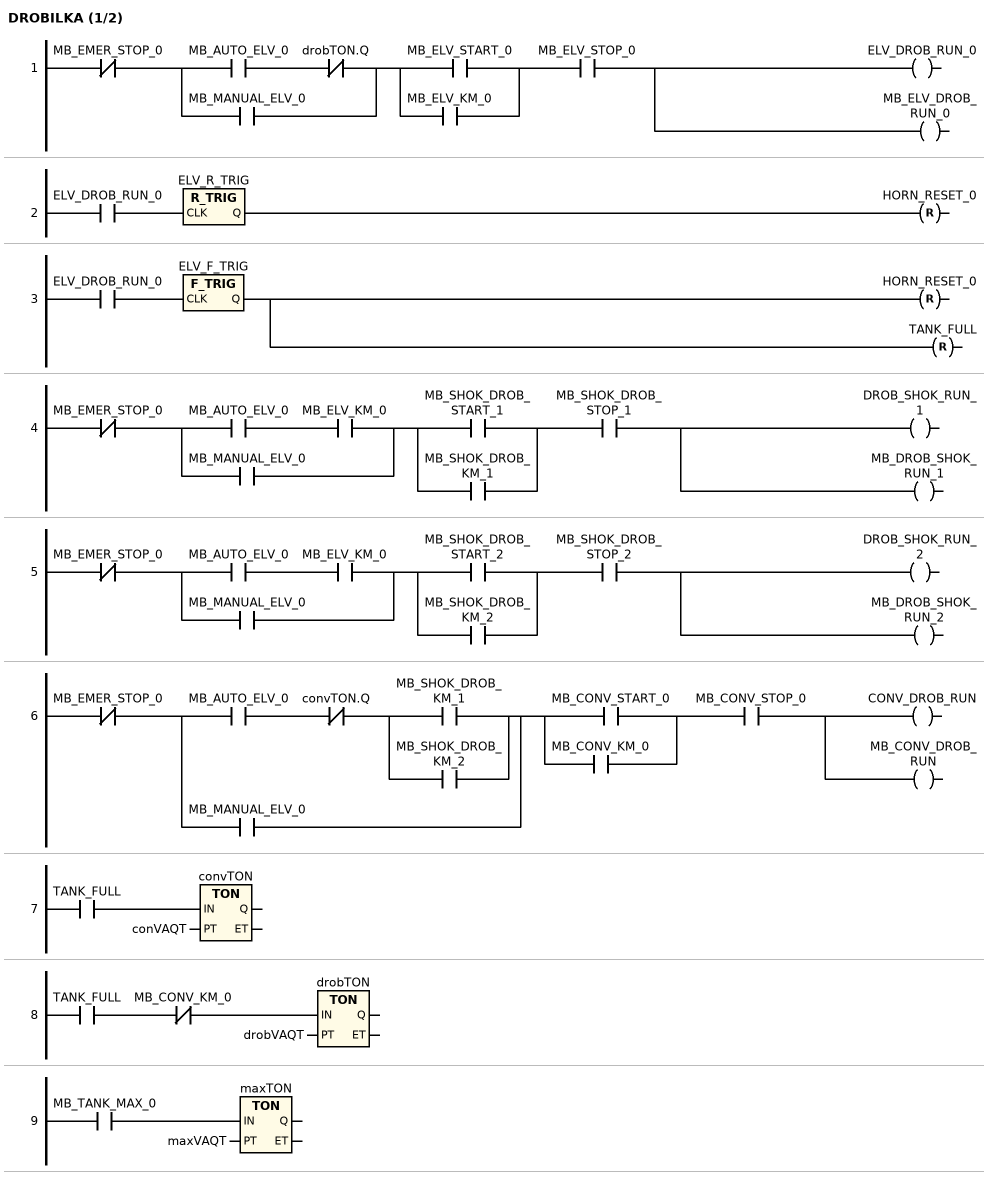
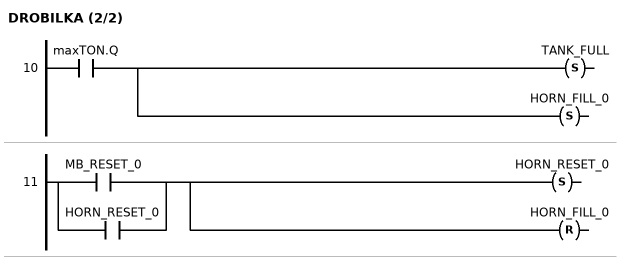
_LD_ (* Ladder Diagram *)
NETWORK 1
	[/MB_EMER_STOP_0] - { [MB_AUTO_ELV_0] - [/drobTON.Q] | [MB_MANUAL_ELV_0] } - { [MB_ELV_START_0] | [MB_ELV_KM_0] } - [MB_ELV_STOP_0] --- (ELV_DROB_RUN_0) (MB_ELV_DROB_RUN_0)
NETWORK 2
	[ELV_DROB_RUN_0] - ELV_R_TRIG:R_TRIG(CLK: *) --- (R HORN_RESET_0)
NETWORK 3
	[ELV_DROB_RUN_0] - ELV_F_TRIG:F_TRIG(CLK: *) --- (R HORN_RESET_0) (R TANK_FULL)
NETWORK 4
	[/MB_EMER_STOP_0] - { [MB_AUTO_ELV_0] - [MB_ELV_KM_0] | [MB_MANUAL_ELV_0] } - { [MB_SHOK_DROB_START_1] | [MB_SHOK_DROB_KM_1] } - [MB_SHOK_DROB_STOP_1] --- (DROB_SHOK_RUN_1) (MB_DROB_SHOK_RUN_1)
NETWORK 5
	[/MB_EMER_STOP_0] - { [MB_AUTO_ELV_0] - [MB_ELV_KM_0] | [MB_MANUAL_ELV_0] } - { [MB_SHOK_DROB_START_2] | [MB_SHOK_DROB_KM_2] } - [MB_SHOK_DROB_STOP_2] --- (DROB_SHOK_RUN_2) (MB_DROB_SHOK_RUN_2)
NETWORK 6
	[/MB_EMER_STOP_0] - { [MB_AUTO_ELV_0] - [/convTON.Q] - { [MB_SHOK_DROB_KM_1] | [MB_SHOK_DROB_KM_2] } | [MB_MANUAL_ELV_0] } - { [MB_CONV_START_0] | [MB_CONV_KM_0] } - [MB_CONV_STOP_0] --- (CONV_DROB_RUN) (MB_CONV_DROB_RUN)
NETWORK 7
	[TANK_FULL] - convTON:TON(IN: *, PT: conVAQT)
NETWORK 8
	[TANK_FULL] - [/MB_CONV_KM_0] - drobTON:TON(IN: *, PT: drobVAQT)
NETWORK 9
	[MB_TANK_MAX_0] - maxTON:TON(IN: *, PT: maxVAQT)
NETWORK 10
	[maxTON.Q] --- (S TANK_FULL) (S HORN_FILL_0)
NETWORK 11
	{ [MB_RESET_0] | [HORN_RESET_0] } --- (S HORN_RESET_0) (R HORN_FILL_0)
_END_LD_
(* the same logic as Structured Text *)
(* Network 1 *)
ELV_DROB_RUN_0 := NOT MB_EMER_STOP_0 AND (MB_AUTO_ELV_0 AND NOT drobTON.Q OR MB_MANUAL_ELV_0) AND (MB_ELV_START_0 OR MB_ELV_KM_0) AND MB_ELV_STOP_0;
MB_ELV_DROB_RUN_0 := ELV_DROB_RUN_0;
(* Network 2 *)
ELV_R_TRIG(CLK := ELV_DROB_RUN_0);
IF ELV_R_TRIG.Q THEN HORN_RESET_0 := FALSE; END_IF;
(* Network 3 *)
ELV_F_TRIG(CLK := ELV_DROB_RUN_0);
IF ELV_F_TRIG.Q THEN HORN_RESET_0 := FALSE; TANK_FULL := FALSE; END_IF;
(* Network 4 *)
DROB_SHOK_RUN_1 := NOT MB_EMER_STOP_0 AND (MB_AUTO_ELV_0 AND MB_ELV_KM_0 OR MB_MANUAL_ELV_0) AND (MB_SHOK_DROB_START_1 OR MB_SHOK_DROB_KM_1) AND MB_SHOK_DROB_STOP_1;
MB_DROB_SHOK_RUN_1 := DROB_SHOK_RUN_1;
(* Network 5 *)
DROB_SHOK_RUN_2 := NOT MB_EMER_STOP_0 AND (MB_AUTO_ELV_0 AND MB_ELV_KM_0 OR MB_MANUAL_ELV_0) AND (MB_SHOK_DROB_START_2 OR MB_SHOK_DROB_KM_2) AND MB_SHOK_DROB_STOP_2;
MB_DROB_SHOK_RUN_2 := DROB_SHOK_RUN_2;
(* Network 6 *)
CONV_DROB_RUN := NOT MB_EMER_STOP_0 AND (MB_AUTO_ELV_0 AND NOT convTON.Q AND (MB_SHOK_DROB_KM_1 OR MB_SHOK_DROB_KM_2) OR MB_MANUAL_ELV_0) AND (MB_CONV_START_0 OR MB_CONV_KM_0) AND MB_CONV_STOP_0;
MB_CONV_DROB_RUN := CONV_DROB_RUN;
(* Network 7 *)
convTON(IN := TANK_FULL, PT := conVAQT);
(* Network 8 *)
drobTON(IN := TANK_FULL AND NOT MB_CONV_KM_0, PT := drobVAQT);
(* Network 9 *)
maxTON(IN := MB_TANK_MAX_0, PT := maxVAQT);
(* Network 10 *)
IF maxTON.Q THEN TANK_FULL := TRUE; HORN_FILL_0 := TRUE; END_IF;
(* Network 11 *)
_p1 := MB_RESET_0 OR HORN_RESET_0;
IF _p1 THEN HORN_RESET_0 := TRUE; HORN_FILL_0 := FALSE; END_IF;
END_PROGRAM

(* POU A_CONVER, CFC *)
FUNCTION_BLOCK A_CONVER
VAR_INPUT
	IN : REAL;
END_VAR
VAR_OUTPUT
	OUT : REAL;

END_VAR
VAR
	LIN1: LIN_TRAFO;
	IN_MIN : REAL := 4;
	IN_MAX : REAL := 20;

END_VAR
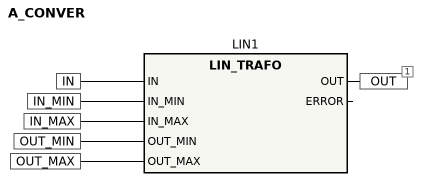
_CFC_ (* Continuous Function Chart, elements in execution order *)
#0 LIN1:LIN_TRAFO(IN: IN, IN_MIN: IN_MIN, IN_MAX: IN_MAX, OUT_MIN: OUT_MIN, OUT_MAX: OUT_MAX)
#1 OUT <= #0.OUT
_END_CFC_
(* the same logic as Structured Text *)
LIN1(IN := IN, IN_MIN := IN_MIN, IN_MAX := IN_MAX, OUT_MIN := OUT_MIN, OUT_MAX := OUT_MAX);
OUT := LIN1.OUT;
END_FUNCTION_BLOCK

(* POU INDUKTIV_2, CFC *)
FUNCTION_BLOCK INDUKTIV_2
VAR_IN_OUT

	(*RESET : BOOL;*)

END_VAR
VAR_INPUT
	START : BOOL;
	kirish : BOOL;
	vaqtIndukt : WORD := 15;
END_VAR

VAR_OUTPUT

	OUT : BOOL;
	ALARM : BOOL;
END_VAR
VAR
	ton1: TON;
	vaqt : TIME;
	ton2: TON;
	TP1: TP;
	TP2: TP;


END_VAR
VAR (* helpers for the ST form of the networks *)
	_t11 : BOOL;
	_t41 : BOOL;
	_t47 : BOOL;
	_t44 : BOOL;
	_t45 : BOOL;
	_en19 : BOOL;
END_VAR
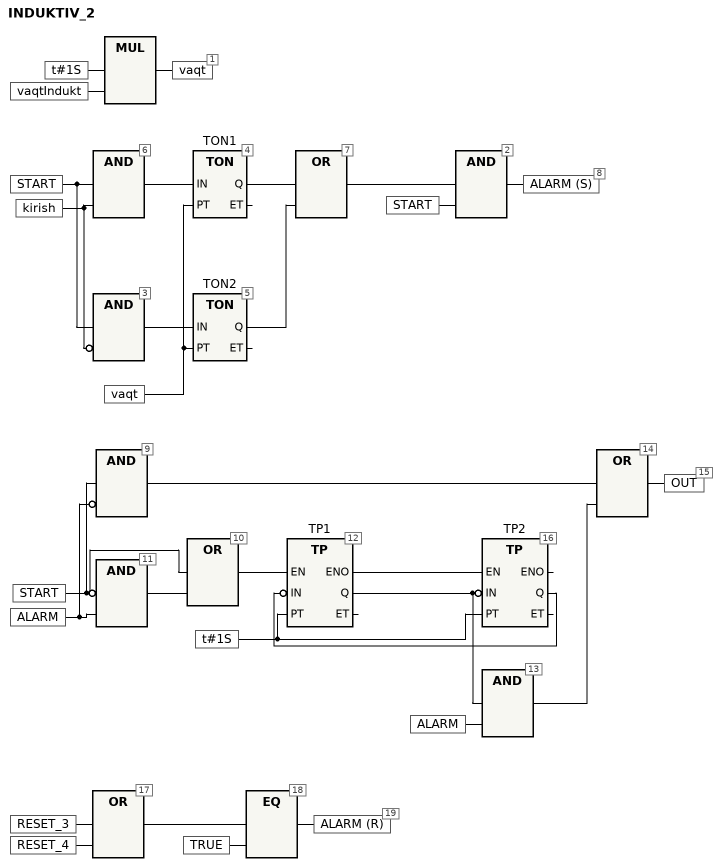
_CFC_ (* Continuous Function Chart, elements in execution order *)
#0 MUL(t#1S, vaqtIndukt)
#1 vaqt <= #0
#2 AND(#7, START)
#3 AND(START, NOT kirish)
#4 TON1:TON(IN: #6, PT: vaqt)
#5 TON2:TON(IN: #3, PT: vaqt)
#6 AND(START, kirish)
#7 OR(#4.Q, #5.Q)
#8 S ALARM <= #2
#9 AND(START, NOT ALARM)
#10 OR(START, #11)
#11 AND(NOT START, ALARM)
#12 TP1:TP(EN: #10, IN: NOT #16.Q, PT: t#1S)
#13 AND(#12.Q, ALARM)
#14 OR(#9, #13)
#15 OUT <= #14
#16 TP2:TP(EN: #12.ENO, IN: NOT #12.Q, PT: t#1S)
#17 OR(RESET_3, RESET_4)
#18 EQ(#17, TRUE)
#19 R ALARM <= #18
_END_CFC_
(* the same logic as Structured Text *)
vaqt := t#1S * vaqtIndukt;
_t41 := _t11 AND START;
TON1(IN := _t47, PT := vaqt);
TON2(IN := START AND NOT kirish, PT := vaqt);
_t47 := START AND kirish;
_t11 := TON1.Q OR TON2.Q;
IF _t41 THEN ALARM := TRUE; END_IF;
_t45 := START OR _t44;
_t44 := NOT START AND ALARM;
_en19 := _t45;
IF _en19 THEN TP1(IN := NOT TP2.Q, PT := t#1S); END_IF;
OUT := (START AND NOT ALARM) OR (TP1.Q AND ALARM);
IF _en19 THEN TP2(IN := NOT TP1.Q, PT := t#1S); END_IF;
IF (RESET_3 OR RESET_4) = TRUE THEN ALARM := FALSE; END_IF;
END_FUNCTION_BLOCK
